LIN {X 0,Y 634.737,Z 843.139,A -85,B 0,C 180,E1 28393.414,E2 28393.414} C_VEL
LIN {X 0,Y 633.485,Z 864.639,A -85,B 0,C 180,E1 28392.949,E2 28392.949} C_VEL
LIN {X 0,Y 631.948,Z 886.443,A -85,B 0,C 180,E1 28392.362,E2 28392.362} C_VEL
LIN {X 0,Y 629.85,Z 912.243,A -85,B 0,C 180,E1 28391.511,E2 28391.511} C_VEL
LIN {X 0,Y 627.434,Z 937.199,A -85,B 0,C 180,E1 28390.495,E2 28390.495} C_VEL
LIN {X 0,Y 625.26,Z 957.685,A -85,B 0,C 180,E1 28389.527,E2 28389.527} C_VEL
LIN {X 0,Y 623.096,Z 976.739,A -85,B 0,C 180,E1 28388.507,E2 28388.507} C_VEL
LIN {X 0,Y 620.859,Z 995.438,A -85,B 0,C 180,E1 28387.383,E2 28387.383} C_VEL
LIN {X 0,Y 618.34,Z 1015.935,A -85,B 0,C 180,E1 28386,E2 28386} C_VEL
LIN {X 0,Y 615.314,Z 1039.357,A -85,B 0,C 180,E1 28384.195,E2 28384.195} C_VEL
LIN {X 0,Y 612.99,Z 1057.389,A -85,B 0,C 180,E1 28382.621,E2 28382.621} C_VEL
LIN {X 0,Y 610.906,Z 1073.81,A -85,B 0,C 180,E1 28381.035,E2 28381.035} C_VEL
LIN {X 0,Y 608.727,Z 1091.946,A -85,B 0,C 180,E1 28379.089,E2 28379.089} C_VEL
LIN {X 0,Y 606.52,Z 1110.307,A -85,B 0,C 180,E1 28376.852,E2 28376.852} C_VEL
LIN {X 0,Y 604.947,Z 1124.916,A -85,B 0,C 180,E1 28374.848,E2 28374.848} C_VEL
LIN {X 0,Y 603.439,Z 1140.182,A -85,B 0,C 180,E1 28372.504,E2 28372.504} C_VEL
LIN {X 0,Y 602.196,Z 1154.243,A -85,B 0,C 180,E1 28370.001,E2 28370.001} C_VEL
LIN {X 0,Y 601.435,Z 1164.532,A -85,B 0,C 180,E1 28367.912,E2 28367.912} C_VEL
LIN {X 0,Y 600.808,Z 1174.331,A -85,B 0,C 180,E1 28365.64,E2 28365.64} C_VEL
LIN {X 0,Y 600.353,Z 1184.273,A -85,B 0,C 180,E1 28362.895,E2 28362.895} C_VEL
LIN {X 0,Y 600.109,Z 1191.1,A -85,B 0,C 180,E1 28360.561,E2 28360.561} C_VEL
LIN {X 0,Y 599.988,Z 1196.552,A -85,B 0,C 180,E1 28358.24,E2 28358.24} C_VEL
LIN {X 0,Y 599.931,Z 1201.053,A -85,B 0,C 180,E1 28355.643,E2 28355.643} C_VEL
LIN {X 0,Y 599.918,Z 1203.723,A -85,B 0,C 180,E1 28353.153,E2 28353.153} C_VEL
LIN {X 0,Y 599.912,Z 1204.759,A -85,B 0,C 180,E1 28351.051,E2 28351.051} C_VEL
LIN {X 0,Y 599.908,Z 1204.782,A -85,B 0,C 180,E1 28349.045,E2 28349.045} C_VEL
LIN {X 0,Y 599.918,Z 1203.791,A -85,B 0,C 180,E1 28346.943,E2 28346.943} C_VEL
LIN {X 0,Y 599.93,Z 1201.177,A -85,B 0,C 180,E1 28344.453,E2 28344.453} C_VEL
LIN {X 0,Y 599.985,Z 1196.758,A -85,B 0,C 180,E1 28341.857,E2 28341.857} C_VEL
LIN {X 0,Y 600.104,Z 1191.355,A -85,B 0,C 180,E1 28339.537,E2 28339.537} C_VEL
LIN {X 0,Y 600.338,Z 1184.575,A -85,B 0,C 180,E1 28337.202,E2 28337.202} C_VEL
LIN {X 0,Y 600.787,Z 1174.735,A -85,B 0,C 180,E1 28334.458,E2 28334.458} C_VEL
LIN {X 0,Y 601.405,Z 1164.995,A -85,B 0,C 180,E1 28332.187,E2 28332.187} C_VEL
LIN {X 0,Y 602.16,Z 1154.762,A -85,B 0,C 180,E1 28330.099,E2 28330.099} C_VEL
LIN {X 0,Y 603.269,Z 1141.958,A -85,B 0,C 180,E1 28327.797,E2 28327.797} C_VEL
LIN {X 0,Y 604.785,Z 1126.491,A -85,B 0,C 180,E1 28325.379,E2 28325.379} C_VEL
LIN {X 0,Y 606.34,Z 1111.848,A -85,B 0,C 180,E1 28323.351,E2 28323.351} C_VEL
LIN {X 0,Y 608.291,Z 1095.443,A -85,B 0,C 180,E1 28321.317,E2 28321.317} C_VEL
LIN {X 0,Y 610.668,Z 1075.839,A -85,B 0,C 180,E1 28319.171,E2 28319.171} C_VEL
LIN {X 0,Y 612.801,Z 1058.916,A -85,B 0,C 180,E1 28317.52,E2 28317.52} C_VEL
LIN {X 0,Y 615.004,Z 1041.616,A -85,B 0,C 180,E1 28315.995,E2 28315.995} C_VEL
LIN {X 0,Y 617.903,Z 1019.546,A -85,B 0,C 180,E1 28314.257,E2 28314.257} C_VEL
LIN {X 0,Y 620.763,Z 996.244,A -85,B 0,C 180,E1 28312.669,E2 28312.669} C_VEL
LIN {X 0,Y 622.991,Z 977.642,A -85,B 0,C 180,E1 28311.544,E2 28311.544} C_VEL
LIN {X 0,Y 625.147,Z 958.697,A -85,B 0,C 180,E1 28310.524,E2 28310.524} C_VEL
LIN {X 0,Y 627.185,Z 939.467,A -85,B 0,C 180,E1 28309.606,E2 28309.606} C_VEL
LIN {X 0,Y 629.333,Z 917.449,A -85,B 0,C 180,E1 28308.69,E2 28308.69} C_VEL
LIN {X 0,Y 631.745,Z 889.26,A -85,B 0,C 180,E1 28307.721,E2 28307.721} C_VEL
LIN {X 0,Y 633.4,Z 865.996,A -85,B 0,C 180,E1 28307.084,E2 28307.084} C_VEL
LIN {X 0,Y 634.659,Z 844.673,A -85,B 0,C 180,E1 28306.616,E2 28306.616} C_VEL
LIN {X 0,Y 635.658,Z 822.464,A -85,B 0,C 180,E1 28306.243,E2 28306.243} C_VEL
LIN {X 0,Y 639.154,Z 652.16,A -85,B 0,C 180,E1 28303.959,E2 28303.959} C_VEL
LIN {X 0,Y 643.512,Z 444.13,A -85,B 0,C 180,E1 28301.119,E2 28301.119} C_VEL
LIN {X 0,Y 644.588,Z 389.647,A -85,B 0,C 180,E1 28300.345,E2 28300.345} C_VEL
LIN {X 0,Y 641.019,Z 373.12,A -85,B 0,C 180,E1 28299.728,E2 28299.728} C_VEL
LIN {X 0,Y 624.364,Z 349.234,A -85,B 0,C 180,E1 28297.601,E2 28297.601} C_VEL
LIN {X 0,Y 614.656,Z 330.629,A -85,B 0,C 180,E1 28295.047,E2 28295.047} C_VEL
LIN {X 0,Y 608.064,Z 317.988,A -85,B 0,C 180,E1 28293.201,E2 28293.201} C_VEL
LIN {X 0,Y 605.38,Z 313.033,A -85,B 0,C 180,E1 28292.438,E2 28292.438} C_VEL
LIN {X 0,Y 603.279,Z 308.898,A -85,B 0,C 180,E1 28291.807,E2 28291.807} C_VEL
LIN {X 0,Y 601.357,Z 305.444,A -85,B 0,C 180,E1 28291.25,E2 28291.25} C_VEL
LIN {X 0,Y 601.143,Z 304.451,A -85,B 0,C 180,E1 28291.04,E2 28291.04} C_VEL
LIN {X 0,Y 601.114,Z 304.316,A -85,B 0,C 180,E1 28287.867,E2 28287.867} C_VEL
LIN {X 0,Y 601.122,Z 304.35,A -85,B 0,C 180,E1 28284.677,E2 28284.677} C_VEL
LIN {X 0,Y 601.115,Z 304.302,A -85,B 0,C 180,E1 28281.466,E2 28281.466} C_VEL
LIN {X 0,Y 601.127,Z 304.348,A -85,B 0,C 180,E1 28278.241,E2 28278.241} C_VEL
LIN {X 0,Y 601.129,Z 304.305,A -85,B 0,C 180,E1 28274.9,E2 28274.9} C_VEL
LIN {X 0,Y 601.127,Z 304.334,A -85,B 0,C 180,E1 28271.611,E2 28271.611} C_VEL
LIN {X 0,Y 601.11,Z 304.31,A -85,B 0,C 180,E1 28268.417,E2 28268.417} C_VEL
LIN {X 0,Y 601.125,Z 304.346,A -85,B 0,C 180,E1 28265.249,E2 28265.249} C_VEL
LIN {X 0,Y 601.113,Z 304.347,A -85,B 0,C 180,E1 28262.097,E2 28262.097} C_VEL
LIN {X 0,Y 601.129,Z 304.354,A -85,B 0,C 180,E1 28258.952,E2 28258.952} C_VEL
LIN {X 0,Y 601.111,Z 304.352,A -85,B 0,C 180,E1 28255.803,E2 28255.803} C_VEL
LIN {X 0,Y 601.138,Z 304.349,A -85,B 0,C 180,E1 28252.545,E2 28252.545} C_VEL
LIN {X 0,Y 601.128,Z 304.345,A -85,B 0,C 180,E1 28249.263,E2 28249.263} C_VEL
LIN {X 0,Y 601.112,Z 304.346,A -85,B 0,C 180,E1 28246.043,E2 28246.043} C_VEL
LIN {X 0,Y 601.134,Z 304.335,A -85,B 0,C 180,E1 28242.878,E2 28242.878} C_VEL
LIN {X 0,Y 601.099,Z 304.343,A -85,B 0,C 180,E1 28239.656,E2 28239.656} C_VEL
LIN {X 0,Y 601.134,Z 304.327,A -85,B 0,C 180,E1 28236.575,E2 28236.575} C_VEL
LIN {X 0,Y 601.094,Z 304.318,A -85,B 0,C 180,E1 28233.418,E2 28233.418} C_VEL
LIN {X 0,Y 601.135,Z 304.326,A -85,B 0,C 180,E1 28230.254,E2 28230.254} C_VEL
LIN {X 0,Y 601.092,Z 304.325,A -85,B 0,C 180,E1 28227.142,E2 28227.142} C_VEL
LIN {X 0,Y 601.126,Z 304.31,A -85,B 0,C 180,E1 28223.926,E2 28223.926} C_VEL
LIN {X 0,Y 601.099,Z 304.355,A -85,B 0,C 180,E1 28220.794,E2 28220.794} C_VEL
LIN {X 0,Y 601.098,Z 304.309,A -85,B 0,C 180,E1 28217.466,E2 28217.466} C_VEL
LIN {X 0,Y 601.112,Z 304.544,A -85,B 0,C 180,E1 28214.878,E2 28214.878} C_VEL
LIN {X 0,Y 602.437,Z 307.817,A -85,B 0,C 180,E1 28214.325,E2 28214.325} C_VEL
LIN {X 0,Y 603.781,Z 310.243,A -85,B 0,C 180,E1 28213.914,E2 28213.914} C_VEL
LIN {X 0,Y 610.058,Z 322.832,A -85,B 0,C 180,E1 28211.917,E2 28211.917} C_VEL
LIN {X 0,Y 618.337,Z 340.119,A -85,B 0,C 180,E1 28209.379,E2 28209.379} C_VEL
LIN {X 0,Y 621.916,Z 347.601,A -85,B 0,C 180,E1 28208.371,E2 28208.371} C_VEL
LIN {X 0,Y 634.739,Z 366.423,A -85,B 0,C 180,E1 28206.763,E2 28206.763} C_VEL
LIN {X 0,Y 635.552,Z 368.337,A -85,B 0,C 180,E1 28206.653,E2 28206.653} C_VEL
LIN {X 0,Y 635.77,Z 369.283,A -85,B 0,C 180,E1 28206.616,E2 28206.616} C_VEL
LIN {X 0,Y 636.509,Z 375.596,A -85,B 0,C 180,E1 28206.442,E2 28206.442} C_VEL
LIN {X 0,Y 635.968,Z 384.479,A -85,B 0,C 180,E1 28206.352,E2 28206.352} C_VEL
LIN {X 0,Y 633.615,Z 401.55,A -85,B 0,C 180,E1 28206.306,E2 28206.306} C_VEL
LIN {X 0,Y 633.425,Z 404.97,A -85,B 0,C 180,E1 28206.27,E2 28206.27} C_VEL
LIN {X 0,Y 627.887,Z 630.342,A -85,B 0,C 180,E1 28203.198,E2 28203.198} C_VEL
LIN {X 0,Y 624.144,Z 782.263,A -85,B 0,C 180,E1 28201.133,E2 28201.133} C_VEL
LIN {X 0,Y 622.848,Z 808.88,A -85,B 0,C 180,E1 28200.626,E2 28200.626} C_VEL
LIN {X 0,Y 621.288,Z 831.683,A -85,B 0,C 180,E1 28200.033,E2 28200.033} C_VEL
LIN {X 0,Y 619.625,Z 852.177,A -85,B 0,C 180,E1 28199.377,E2 28199.377} C_VEL
LIN {X 0,Y 617.403,Z 876.604,A -85,B 0,C 180,E1 28198.43,E2 28198.43} C_VEL
LIN {X 0,Y 615.001,Z 898.626,A -85,B 0,C 180,E1 28197.393,E2 28197.393} C_VEL
LIN {X 0,Y 612.877,Z 916.885,A -85,B 0,C 180,E1 28196.404,E2 28196.404} C_VEL
LIN {X 0,Y 610.566,Z 935.623,A -85,B 0,C 180,E1 28195.251,E2 28195.251} C_VEL
LIN {X 0,Y 607.657,Z 957.975,A -85,B 0,C 180,E1 28193.671,E2 28193.671} C_VEL
LIN {X 0,Y 604.491,Z 983.088,A -85,B 0,C 180,E1 28191.626,E2 28191.626} C_VEL
LIN {X 0,Y 602.054,Z 1002.514,A -85,B 0,C 180,E1 28189.803,E2 28189.803} C_VEL
LIN {X 0,Y 600.17,Z 1018.198,A -85,B 0,C 180,E1 28188.152,E2 28188.152} C_VEL
LIN {X 0,Y 598.217,Z 1035.5,A -85,B 0,C 180,E1 28186.108,E2 28186.108} C_VEL
LIN {X 0,Y 596.541,Z 1050.571,A -85,B 0,C 180,E1 28184.066,E2 28184.066} C_VEL
LIN {X 0,Y 595.307,Z 1063.353,A -85,B 0,C 180,E1 28182.119,E2 28182.119} C_VEL
LIN {X 0,Y 594.083,Z 1077.311,A -85,B 0,C 180,E1 28179.689,E2 28179.689} C_VEL
LIN {X 0,Y 593.289,Z 1087.834,A -85,B 0,C 180,E1 28177.553,E2 28177.553} C_VEL
LIN {X 0,Y 592.738,Z 1096.969,A -85,B 0,C 180,E1 28175.42,E2 28175.42} C_VEL
LIN {X 0,Y 592.306,Z 1106.272,A -85,B 0,C 180,E1 28172.806,E2 28172.806} C_VEL
LIN {X 0,Y 592.077,Z 1112.145,A -85,B 0,C 180,E1 28170.774,E2 28170.774} C_VEL
LIN {X 0,Y 591.987,Z 1116.904,A -85,B 0,C 180,E1 28168.742,E2 28168.742} C_VEL
LIN {X 0,Y 591.917,Z 1121.208,A -85,B 0,C 180,E1 28166.32,E2 28166.32} C_VEL
LIN {X 0,Y 591.912,Z 1123.779,A -85,B 0,C 180,E1 28163.891,E2 28163.891} C_VEL
LIN {X 0,Y 591.915,Z 1124.8,A -85,B 0,C 180,E1 28161.843,E2 28161.843} C_VEL
LIN {X 0,Y 591.904,Z 1124.734,A -85,B 0,C 180,E1 28159.783,E2 28159.783} C_VEL
LIN {X 0,Y 591.918,Z 1123.242,A -85,B 0,C 180,E1 28157.315,E2 28157.315} C_VEL
LIN {X 0,Y 591.921,Z 1120.275,A -85,B 0,C 180,E1 28155.022,E2 28155.022} C_VEL
LIN {X 0,Y 591.988,Z 1116.421,A -85,B 0,C 180,E1 28152.941,E2 28152.941} C_VEL
LIN {X 0,Y 592.112,Z 1111.473,A -85,B 0,C 180,E1 28150.877,E2 28150.877} C_VEL
LIN {X 0,Y 592.395,Z 1103.669,A -85,B 0,C 180,E1 28148.307,E2 28148.307} C_VEL
LIN {X 0,Y 592.828,Z 1095.329,A -85,B 0,C 180,E1 28146.088,E2 28146.088} C_VEL
LIN {X 0,Y 593.414,Z 1086.275,A -85,B 0,C 180,E1 28144.018,E2 28144.018} C_VEL
LIN {X 0,Y 594.431,Z 1073.185,A -85,B 0,C 180,E1 28141.465,E2 28141.465} C_VEL
LIN {X 0,Y 595.521,Z 1061.026,A -85,B 0,C 180,E1 28139.421,E2 28139.421} C_VEL
LIN {X 0,Y 596.932,Z 1047.21,A -85,B 0,C 180,E1 28137.361,E2 28137.361} C_VEL
LIN {X 0,Y 598.756,Z 1030.354,A -85,B 0,C 180,E1 28135.173,E2 28135.173} C_VEL
LIN {X 0,Y 600.547,Z 1015.057,A -85,B 0,C 180,E1 28133.413,E2 28133.413} C_VEL
LIN {X 0,Y 602.877,Z 996.133,A -85,B 0,C 180,E1 28131.476,E2 28131.476} C_VEL
LIN {X 0,Y 605.186,Z 976.858,A -85,B 0,C 180,E1 28129.758,E2 28129.758} C_VEL
LIN {X 0,Y 608.508,Z 951.843,A -85,B 0,C 180,E1 28127.775,E2 28127.775} C_VEL
LIN {X 0,Y 610.992,Z 932.614,A -85,B 0,C 180,E1 28126.453,E2 28126.453} C_VEL
LIN {X 0,Y 613.37,Z 913.498,A -85,B 0,C 180,E1 28125.296,E2 28125.296} C_VEL
LIN {X 0,Y 616.143,Z 889.259,A -85,B 0,C 180,E1 28124.037,E2 28124.037} C_VEL
LIN {X 0,Y 618.322,Z 867.895,A -85,B 0,C 180,E1 28123.105,E2 28123.105} C_VEL
LIN {X 0,Y 620.368,Z 845.635,A -85,B 0,C 180,E1 28122.287,E2 28122.287} C_VEL
LIN {X 0,Y 622.332,Z 819.853,A -85,B 0,C 180,E1 28121.532,E2 28121.532} C_VEL
LIN {X 0,Y 623.576,Z 798.797,A -85,B 0,C 180,E1 28121.052,E2 28121.052} C_VEL
LIN {X 0,Y 624.552,Z 776.726,A -85,B 0,C 180,E1 28120.672,E2 28120.672} C_VEL
LIN {X 0,Y 630.566,Z 536.64,A -85,B 0,C 180,E1 28117.405,E2 28117.405} C_VEL
LIN {X 0,Y 634.45,Z 387.315,A -85,B 0,C 180,E1 28115.324,E2 28115.324} C_VEL
LIN {X 0,Y 631.23,Z 372.127,A -85,B 0,C 180,E1 28114.713,E2 28114.713} C_VEL
LIN {X 0,Y 621.138,Z 357.085,A -85,B 0,C 180,E1 28113.294,E2 28113.294} C_VEL
LIN {X 0,Y 614.055,Z 346.626,A -85,B 0,C 180,E1 28112.172,E2 28112.172} C_VEL
LIN {X 0,Y 607.583,Z 333.131,A -85,B 0,C 180,E1 28109.91,E2 28109.91} C_VEL
LIN {X 0,Y 602.57,Z 323.528,A -85,B 0,C 180,E1 28108.116,E2 28108.116} C_VEL
LIN {X 0,Y 600.308,Z 319.191,A -85,B 0,C 180,E1 28107.261,E2 28107.261} C_VEL
LIN {X 0,Y 597.846,Z 314.566,A -85,B 0,C 180,E1 28106.308,E2 28106.308} C_VEL
LIN {X 0,Y 595.889,Z 310.557,A -85,B 0,C 180,E1 28105.482,E2 28105.482} C_VEL
LIN {X 0,Y 593.523,Z 306.861,A -85,B 0,C 180,E1 28104.59,E2 28104.59} C_VEL
LIN {X 0,Y 593.205,Z 305.46,A -85,B 0,C 180,E1 28104.235,E2 28104.235} C_VEL
LIN {X 0,Y 593.187,Z 305.301,A -85,B 0,C 180,E1 28100.938,E2 28100.938} C_VEL
LIN {X 0,Y 593.186,Z 305.3,A -85,B 0,C 180,E1 28097.759,E2 28097.759} C_VEL
LIN {X 0,Y 593.181,Z 305.343,A -85,B 0,C 180,E1 28094.546,E2 28094.546} C_VEL
LIN {X 0,Y 593.18,Z 305.301,A -85,B 0,C 180,E1 28091.375,E2 28091.375} C_VEL
LIN {X 0,Y 593.176,Z 305.313,A -85,B 0,C 180,E1 28088.238,E2 28088.238} C_VEL
LIN {X 0,Y 593.18,Z 305.328,A -85,B 0,C 180,E1 28085.029,E2 28085.029} C_VEL
LIN {X 0,Y 593.179,Z 305.295,A -85,B 0,C 180,E1 28081.835,E2 28081.835} C_VEL
LIN {X 0,Y 593.193,Z 305.339,A -85,B 0,C 180,E1 28078.551,E2 28078.551} C_VEL
LIN {X 0,Y 593.184,Z 305.298,A -85,B 0,C 180,E1 28075.262,E2 28075.262} C_VEL
LIN {X 0,Y 593.186,Z 305.314,A -85,B 0,C 180,E1 28072.055,E2 28072.055} C_VEL
LIN {X 0,Y 593.178,Z 305.326,A -85,B 0,C 180,E1 28068.818,E2 28068.818} C_VEL
LIN {X 0,Y 593.18,Z 305.296,A -85,B 0,C 180,E1 28065.653,E2 28065.653} C_VEL
LIN {X 0,Y 593.178,Z 305.34,A -85,B 0,C 180,E1 28062.438,E2 28062.438} C_VEL
LIN {X 0,Y 593.19,Z 305.307,A -85,B 0,C 180,E1 28059.166,E2 28059.166} C_VEL
LIN {X 0,Y 593.186,Z 305.296,A -85,B 0,C 180,E1 28055.926,E2 28055.926} C_VEL
LIN {X 0,Y 593.181,Z 305.318,A -85,B 0,C 180,E1 28052.601,E2 28052.601} C_VEL
LIN {X 0,Y 593.233,Z 305.627,A -85,B 0,C 180,E1 28051.214,E2 28051.214} C_VEL
LIN {X 0,Y 594.731,Z 309.137,A -85,B 0,C 180,E1 28050.488,E2 28050.488} C_VEL
LIN {X 0,Y 596.204,Z 311.055,A -85,B 0,C 180,E1 28050.015,E2 28050.015} C_VEL
LIN {X 0,Y 598.26,Z 314.959,A -85,B 0,C 180,E1 28049.241,E2 28049.241} C_VEL
LIN {X 0,Y 599.372,Z 316.945,A -85,B 0,C 180,E1 28048.845,E2 28048.845} C_VEL
LIN {X 0,Y 602.237,Z 322.081,A -85,B 0,C 180,E1 28047.857,E2 28047.857} C_VEL
LIN {X 0,Y 605.079,Z 327.328,A -85,B 0,C 180,E1 28046.907,E2 28046.907} C_VEL
LIN {X 0,Y 609.467,Z 335.318,A -85,B 0,C 180,E1 28045.528,E2 28045.528} C_VEL
LIN {X 0,Y 615.852,Z 348.153,A -85,B 0,C 180,E1 28043.542,E2 28043.542} C_VEL
LIN {X 0,Y 617.493,Z 350.954,A -85,B 0,C 180,E1 28043.192,E2 28043.192} C_VEL
LIN {X 0,Y 633.776,Z 374.667,A -85,B 0,C 180,E1 28040.944,E2 28040.944} C_VEL
LIN {X 0,Y 636.298,Z 378.781,A -85,B 0,C 180,E1 28040.613,E2 28040.613} C_VEL
LIN {X 0,Y 639.01,Z 393.151,A -85,B 0,C 180,E1 28040.1,E2 28040.1} C_VEL
LIN {X 0,Y 634.195,Z 606.611,A -85,B 0,C 180,E1 28037.148,E2 28037.148} C_VEL
LIN {X 0,Y 629.632,Z 823.84,A -85,B 0,C 180,E1 28034.222,E2 28034.222} C_VEL
LIN {X 0,Y 628.645,Z 846.019,A -85,B 0,C 180,E1 28033.849,E2 28033.849} C_VEL
LIN {X 0,Y 627.348,Z 868.333,A -85,B 0,C 180,E1 28033.359,E2 28033.359} C_VEL
LIN {X 0,Y 625.389,Z 894.349,A -85,B 0,C 180,E1 28032.622,E2 28032.622} C_VEL
LIN {X 0,Y 623.049,Z 919.238,A -85,B 0,C 180,E1 28031.733,E2 28031.733} C_VEL
LIN {X 0,Y 620.978,Z 939.457,A -85,B 0,C 180,E1 28030.883,E2 28030.883} C_VEL
LIN {X 0,Y 618.822,Z 958.686,A -85,B 0,C 180,E1 28029.96,E2 28029.96} C_VEL
LIN {X 0,Y 616.544,Z 977.636,A -85,B 0,C 180,E1 28028.933,E2 28028.933} C_VEL
LIN {X 0,Y 614.088,Z 997.058,A -85,B 0,C 180,E1 28027.749,E2 28027.749} C_VEL
LIN {X 0,Y 610.965,Z 1020.889,A -85,B 0,C 180,E1 28026.097,E2 28026.097} C_VEL
LIN {X 0,Y 608.094,Z 1041.617,A -85,B 0,C 180,E1 28024.446,E2 28024.446} C_VEL
LIN {X 0,Y 605.719,Z 1059.052,A -85,B 0,C 180,E1 28022.894,E2 28022.894} C_VEL
LIN {X 0,Y 603.289,Z 1077.265,A -85,B 0,C 180,E1 28021.092,E2 28021.092} C_VEL
LIN {X 0,Y 600.702,Z 1097.146,A -85,B 0,C 180,E1 28018.862,E2 28018.862} C_VEL
LIN {X 0,Y 598.746,Z 1112.644,A -85,B 0,C 180,E1 28016.903,E2 28016.903} C_VEL
LIN {X 0,Y 597.075,Z 1127.449,A -85,B 0,C 180,E1 28014.815,E2 28014.815} C_VEL
LIN {X 0,Y 595.364,Z 1143.703,A -85,B 0,C 180,E1 28012.202,E2 28012.202} C_VEL
LIN {X 0,Y 594.298,Z 1155.27,A -85,B 0,C 180,E1 28010.073,E2 28010.073} C_VEL
LIN {X 0,Y 593.5,Z 1165.448,A -85,B 0,C 180,E1 28007.957,E2 28007.957} C_VEL
LIN {X 0,Y 592.788,Z 1176.306,A -85,B 0,C 180,E1 28005.356,E2 28005.356} C_VEL
LIN {X 0,Y 592.348,Z 1185.179,A -85,B 0,C 180,E1 28002.775,E2 28002.775} C_VEL
LIN {X 0,Y 592.108,Z 1191.86,A -85,B 0,C 180,E1 28000.41,E2 28000.41} C_VEL
LIN {X 0,Y 591.981,Z 1197.542,A -85,B 0,C 180,E1 27997.863,E2 27997.863} C_VEL
LIN {X 0,Y 591.928,Z 1201.66,A -85,B 0,C 180,E1 27995.234,E2 27995.234} C_VEL
LIN {X 0,Y 591.915,Z 1203.925,A -85,B 0,C 180,E1 27992.905,E2 27992.905} C_VEL
LIN {X 0,Y 591.895,Z 1204.849,A -85,B 0,C 180,E1 27990.678,E2 27990.678} C_VEL
LIN {X 0,Y 591.908,Z 1204.623,A -85,B 0,C 180,E1 27988.355,E2 27988.355} C_VEL
LIN {X 0,Y 591.918,Z 1202.789,A -85,B 0,C 180,E1 27985.738,E2 27985.738} C_VEL
LIN {X 0,Y 591.944,Z 1199.546,A -85,B 0,C 180,E1 27983.307,E2 27983.307} C_VEL
LIN {X 0,Y 592.022,Z 1195.103,A -85,B 0,C 180,E1 27980.963,E2 27980.963} C_VEL
LIN {X 0,Y 592.224,Z 1188.471,A -85,B 0,C 180,E1 27978.31,E2 27978.31} C_VEL
LIN {X 0,Y 592.556,Z 1180.571,A -85,B 0,C 180,E1 27975.838,E2 27975.838} C_VEL
LIN {X 0,Y 593.028,Z 1172.305,A -85,B 0,C 180,E1 27973.646,E2 27973.646} C_VEL
LIN {X 0,Y 593.709,Z 1162.694,A -85,B 0,C 180,E1 27971.44,E2 27971.44} C_VEL
LIN {X 0,Y 594.841,Z 1149.447,A -85,B 0,C 180,E1 27968.815,E2 27968.815} C_VEL
LIN {X 0,Y 596.107,Z 1136.315,A -85,B 0,C 180,E1 27966.567,E2 27966.567} C_VEL
LIN {X 0,Y 597.54,Z 1122.985,A -85,B 0,C 180,E1 27964.53,E2 27964.53} C_VEL
LIN {X 0,Y 599.573,Z 1106.413,A -85,B 0,C 180,E1 27962.273,E2 27962.273} C_VEL
LIN {X 0,Y 601.819,Z 1088.229,A -85,B 0,C 180,E1 27960.105,E2 27960.105} C_VEL
LIN {X 0,Y 603.941,Z 1072.291,A -85,B 0,C 180,E1 27958.4,E2 27958.4} C_VEL
LIN {X 0,Y 606.351,Z 1054.613,A -85,B 0,C 180,E1 27956.694,E2 27956.694} C_VEL
LIN {X 0,Y 609.496,Z 1031.566,A -85,B 0,C 180,E1 27954.729,E2 27954.729} C_VEL
LIN {X 0,Y 612.158,Z 1011.517,A -85,B 0,C 180,E1 27953.229,E2 27953.229} C_VEL
LIN {X 0,Y 614.692,Z 992.1,A -85,B 0,C 180,E1 27951.934,E2 27951.934} C_VEL
LIN {X 0,Y 617.675,Z 968.571,A -85,B 0,C 180,E1 27950.549,E2 27950.549} C_VEL
LIN {X 0,Y 620.471,Z 943.985,A -85,B 0,C 180,E1 27949.32,E2 27949.32} C_VEL
LIN {X 0,Y 622.709,Z 922.583,A -85,B 0,C 180,E1 27948.399,E2 27948.399} C_VEL
LIN {X 0,Y 624.663,Z 901.901,A -85,B 0,C 180,E1 27947.634,E2 27947.634} C_VEL
LIN {X 0,Y 626.529,Z 879.6,A -85,B 0,C 180,E1 27946.939,E2 27946.939} C_VEL
LIN {X 0,Y 628.34,Z 852.631,A -85,B 0,C 180,E1 27946.278,E2 27946.278} C_VEL
LIN {X 0,Y 629.539,Z 827.007,A -85,B 0,C 180,E1 27945.822,E2 27945.822} C_VEL
LIN {X 0,Y 632.652,Z 684.755,A -85,B 0,C 180,E1 27943.901,E2 27943.901} C_VEL
LIN {X 0,Y 637.392,Z 469.924,A -85,B 0,C 180,E1 27940.958,E2 27940.958} C_VEL
LIN {X 0,Y 639.12,Z 391.738,A -85,B 0,C 180,E1 27939.848,E2 27939.848} C_VEL
LIN {X 0,Y 636.184,Z 378.113,A -85,B 0,C 180,E1 27939.33,E2 27939.33} C_VEL
LIN {X 0,Y 616.066,Z 349.467,A -85,B 0,C 180,E1 27936.733,E2 27936.733} C_VEL
LIN {X 0,Y 606.711,Z 331.431,A -85,B 0,C 180,E1 27934.193,E2 27934.193} C_VEL
LIN {X 0,Y 599.863,Z 318.515,A -85,B 0,C 180,E1 27932.235,E2 27932.235} C_VEL
LIN {X 0,Y 597.671,Z 314.326,A -85,B 0,C 180,E1 27931.577,E2 27931.577} C_VEL
LIN {X 0,Y 595.189,Z 309.685,A -85,B 0,C 180,E1 27930.823,E2 27930.823} C_VEL
LIN {X 0,Y 593.374,Z 306.265,A -85,B 0,C 180,E1 27930.255,E2 27930.255} C_VEL
LIN {X 0,Y 593.197,Z 305.427,A -85,B 0,C 180,E1 27930.041,E2 27930.041} C_VEL
LIN {X 0,Y 593.181,Z 305.29,A -85,B 0,C 180,E1 27926.856,E2 27926.856} C_VEL
LIN {X 0,Y 593.179,Z 305.331,A -85,B 0,C 180,E1 27923.652,E2 27923.652} C_VEL
LIN {X 0,Y 593.178,Z 305.302,A -85,B 0,C 180,E1 27920.525,E2 27920.525} C_VEL
LIN {X 0,Y 593.18,Z 305.306,A -85,B 0,C 180,E1 27917.359,E2 27917.359} C_VEL
LIN {X 0,Y 593.181,Z 305.315,A -85,B 0,C 180,E1 27914.148,E2 27914.148} C_VEL
LIN {X 0,Y 593.187,Z 305.297,A -85,B 0,C 180,E1 27910.882,E2 27910.882} C_VEL
LIN {X 0,Y 593.192,Z 305.324,A -85,B 0,C 180,E1 27907.555,E2 27907.555} C_VEL
LIN {X 0,Y 593.176,Z 305.33,A -85,B 0,C 180,E1 27904.35,E2 27904.35} C_VEL
LIN {X 0,Y 593.187,Z 305.328,A -85,B 0,C 180,E1 27901.159,E2 27901.159} C_VEL
LIN {X 0,Y 593.17,Z 305.328,A -85,B 0,C 180,E1 27897.971,E2 27897.971} C_VEL
LIN {X 0,Y 593.194,Z 305.332,A -85,B 0,C 180,E1 27894.681,E2 27894.681} C_VEL
LIN {X 0,Y 593.181,Z 305.337,A -85,B 0,C 180,E1 27891.469,E2 27891.469} C_VEL
LIN {X 0,Y 593.177,Z 305.34,A -85,B 0,C 180,E1 27888.132,E2 27888.132} C_VEL
LIN {X 0,Y 593.2,Z 305.338,A -85,B 0,C 180,E1 27884.955,E2 27884.955} C_VEL
LIN {X 0,Y 593.164,Z 305.344,A -85,B 0,C 180,E1 27881.727,E2 27881.727} C_VEL
LIN {X 0,Y 593.199,Z 305.336,A -85,B 0,C 180,E1 27878.499,E2 27878.499} C_VEL
LIN {X 0,Y 593.152,Z 305.29,A -85,B 0,C 180,E1 27875.394,E2 27875.394} C_VEL
LIN {X 0,Y 593.2,Z 305.333,A -85,B 0,C 180,E1 27872.166,E2 27872.166} C_VEL
LIN {X 0,Y 593.157,Z 305.291,A -85,B 0,C 180,E1 27869.06,E2 27869.06} C_VEL
LIN {X 0,Y 593.175,Z 305.345,A -85,B 0,C 180,E1 27865.736,E2 27865.736} C_VEL
LIN {X 0,Y 593.179,Z 305.289,A -85,B 0,C 180,E1 27862.553,E2 27862.553} C_VEL
LIN {X 0,Y 593.153,Z 305.317,A -85,B 0,C 180,E1 27859.336,E2 27859.336} C_VEL
LIN {X 0,Y 593.197,Z 305.323,A -85,B 0,C 180,E1 27856.149,E2 27856.149} C_VEL
LIN {X 0,Y 593.268,Z 305.827,A -85,B 0,C 180,E1 27855.753,E2 27855.753} C_VEL
LIN {X 0,Y 594.698,Z 309.158,A -85,B 0,C 180,E1 27855.194,E2 27855.194} C_VEL
LIN {X 0,Y 595.935,Z 311.517,A -85,B 0,C 180,E1 27854.787,E2 27854.787} C_VEL
LIN {X 0,Y 598.222,Z 315.85,A -85,B 0,C 180,E1 27854.051,E2 27854.051} C_VEL
LIN {X 0,Y 604.443,Z 328.451,A -85,B 0,C 180,E1 27852.033,E2 27852.033} C_VEL
LIN {X 0,Y 612.463,Z 345.252,A -85,B 0,C 180,E1 27849.545,E2 27849.545} C_VEL
LIN {X 0,Y 613.838,Z 347.799,A -85,B 0,C 180,E1 27849.217,E2 27849.217} C_VEL
LIN {X 0,Y 629.897,Z 371.21,A -85,B 0,C 180,E1 27847.167,E2 27847.167} C_VEL
LIN {X 0,Y 630.758,Z 373.41,A -85,B 0,C 180,E1 27847.045,E2 27847.045} C_VEL
LIN {X 0,Y 633.841,Z 388.559,A -85,B 0,C 180,E1 27846.494,E2 27846.494} C_VEL
LIN {X 0,Y 633.425,Z 404.97,A -85,B 0,C 180,E1 27846.27,E2 27846.27} C_VEL
LIN {X 0,Y 632.552,Z 412.675,A -85,B 0,C 180,E1 27846.23,E2 27846.23} C_VEL
LIN {X 0,Y 627.751,Z 433.322,A -85,B 0,C 180,E1 27846.364,E2 27846.364} C_VEL
LIN {X 0,Y 627.068,Z 439.932,A -85,B 0,C 180,E1 27846.324,E2 27846.324} C_VEL
LIN {X 0,Y 621.351,Z 664.116,A -85,B 0,C 180,E1 27843.259,E2 27843.259} C_VEL
LIN {X 0,Y 618.257,Z 782.871,A -85,B 0,C 180,E1 27841.63,E2 27841.63} C_VEL
LIN {X 0,Y 616.874,Z 809.805,A -85,B 0,C 180,E1 27841.111,E2 27841.111} C_VEL
LIN {X 0,Y 615.261,Z 832.313,A -85,B 0,C 180,E1 27840.52,E2 27840.52} C_VEL
LIN {X 0,Y 613.517,Z 852.781,A -85,B 0,C 180,E1 27839.86,E2 27839.86} C_VEL
LIN {X 0,Y 611.188,Z 877.138,A -85,B 0,C 180,E1 27838.909,E2 27838.909} C_VEL
LIN {X 0,Y 608.663,Z 899.206,A -85,B 0,C 180,E1 27837.862,E2 27837.862} C_VEL
LIN {X 0,Y 606.412,Z 917.602,A -85,B 0,C 180,E1 27836.857,E2 27836.857} C_VEL
LIN {X 0,Y 603.904,Z 936.945,A -85,B 0,C 180,E1 27835.655,E2 27835.655} C_VEL
LIN {X 0,Y 600.726,Z 959.903,A -85,B 0,C 180,E1 27834.003,E2 27834.003} C_VEL
LIN {X 0,Y 598.217,Z 977.418,A -85,B 0,C 180,E1 27832.556,E2 27832.556} C_VEL
LIN {X 0,Y 595.281,Z 998.952,A -85,B 0,C 180,E1 27830.551,E2 27830.551} C_VEL
LIN {X 0,Y 593.082,Z 1015.822,A -85,B 0,C 180,E1 27828.784,E2 27828.784} C_VEL
LIN {X 0,Y 591.192,Z 1030.97,A -85,B 0,C 180,E1 27827.013,E2 27827.013} C_VEL
LIN {X 0,Y 589.21,Z 1048.084,A -85,B 0,C 180,E1 27824.746,E2 27824.746} C_VEL
LIN {X 0,Y 587.781,Z 1061.093,A -85,B 0,C 180,E1 27822.776,E2 27822.776} C_VEL
LIN {X 0,Y 586.625,Z 1073.229,A -85,B 0,C 180,E1 27820.707,E2 27820.707} C_VEL
LIN {X 0,Y 585.533,Z 1086.182,A -85,B 0,C 180,E1 27818.148,E2 27818.148} C_VEL
LIN {X 0,Y 584.922,Z 1095.107,A -85,B 0,C 180,E1 27816.084,E2 27816.084} C_VEL
LIN {X 0,Y 584.465,Z 1103.153,A -85,B 0,C 180,E1 27813.924,E2 27813.924} C_VEL
LIN {X 0,Y 584.149,Z 1111.209,A -85,B 0,C 180,E1 27811.275,E2 27811.275} C_VEL
LIN {X 0,Y 584.002,Z 1116.344,A -85,B 0,C 180,E1 27809.117,E2 27809.117} C_VEL
LIN {X 0,Y 583.936,Z 1120.138,A -85,B 0,C 180,E1 27807.055,E2 27807.055} C_VEL
LIN {X 0,Y 583.904,Z 1123.299,A -85,B 0,C 180,E1 27804.596,E2 27804.596} C_VEL
LIN {X 0,Y 583.917,Z 1124.737,A -85,B 0,C 180,E1 27802.126,E2 27802.126} C_VEL
LIN {X 0,Y 583.897,Z 1124.797,A -85,B 0,C 180,E1 27800.04,E2 27800.04} C_VEL
LIN {X 0,Y 583.911,Z 1123.726,A -85,B 0,C 180,E1 27797.901,E2 27797.901} C_VEL
LIN {X 0,Y 583.923,Z 1120.888,A -85,B 0,C 180,E1 27795.32,E2 27795.32} C_VEL
LIN {X 0,Y 583.992,Z 1116.939,A -85,B 0,C 180,E1 27793.079,E2 27793.079} C_VEL
LIN {X 0,Y 584.109,Z 1112.194,A -85,B 0,C 180,E1 27791.02,E2 27791.02} C_VEL
LIN {X 0,Y 584.346,Z 1105.953,A -85,B 0,C 180,E1 27788.836,E2 27788.836} C_VEL
LIN {X 0,Y 584.837,Z 1096.628,A -85,B 0,C 180,E1 27786.204,E2 27786.204} C_VEL
LIN {X 0,Y 585.44,Z 1087.59,A -85,B 0,C 180,E1 27784.074,E2 27784.074} C_VEL
LIN {X 0,Y 586.331,Z 1076.704,A -85,B 0,C 180,E1 27781.844,E2 27781.844} C_VEL
LIN {X 0,Y 587.625,Z 1062.856,A -85,B 0,C 180,E1 27779.419,E2 27779.419} C_VEL
LIN {X 0,Y 588.894,Z 1050.727,A -85,B 0,C 180,E1 27777.551,E2 27777.551} C_VEL
LIN {X 0,Y 590.736,Z 1035.048,A -85,B 0,C 180,E1 27775.399,E2 27775.399} C_VEL
LIN {X 0,Y 592.834,Z 1017.755,A -85,B 0,C 180,E1 27773.341,E2 27773.341} C_VEL
LIN {X 0,Y 594.858,Z 1001.983,A -85,B 0,C 180,E1 27771.667,E2 27771.667} C_VEL
LIN {X 0,Y 598.1,Z 978.43,A -85,B 0,C 180,E1 27769.436,E2 27769.436} C_VEL
LIN {X 0,Y 600.601,Z 961.131,A -85,B 0,C 180,E1 27767.992,E2 27767.992} C_VEL
LIN {X 0,Y 603.69,Z 939.447,A -85,B 0,C 180,E1 27766.402,E2 27766.402} C_VEL
LIN {X 0,Y 606.376,Z 918.942,A -85,B 0,C 180,E1 27765.111,E2 27765.111} C_VEL
LIN {X 0,Y 608.615,Z 900.948,A -85,B 0,C 180,E1 27764.117,E2 27764.117} C_VEL
LIN {X 0,Y 610.995,Z 880.4,A -85,B 0,C 180,E1 27763.126,E2 27763.126} C_VEL
LIN {X 0,Y 613.551,Z 855.071,A -85,B 0,C 180,E1 27762.108,E2 27762.108} C_VEL
LIN {X 0,Y 615.387,Z 833.714,A -85,B 0,C 180,E1 27761.406,E2 27761.406} C_VEL
LIN {X 0,Y 616.889,Z 813.151,A -85,B 0,C 180,E1 27760.856,E2 27760.856} C_VEL
LIN {X 0,Y 618.34,Z 788.047,A -85,B 0,C 180,E1 27760.338,E2 27760.338} C_VEL
LIN {X 0,Y 619.677,Z 742.474,A -85,B 0,C 180,E1 27759.688,E2 27759.688} C_VEL
LIN {X 0,Y 626.063,Z 503.632,A -85,B 0,C 180,E1 27756.407,E2 27756.407} C_VEL
LIN {X 0,Y 629.227,Z 389.301,A -85,B 0,C 180,E1 27754.791,E2 27754.791} C_VEL
LIN {X 0,Y 626.621,Z 376.921,A -85,B 0,C 180,E1 27754.283,E2 27754.283} C_VEL
LIN {X 0,Y 614.739,Z 359.161,A -85,B 0,C 180,E1 27752.546,E2 27752.546} C_VEL
LIN {X 0,Y 606.2,Z 347.127,A -85,B 0,C 180,E1 27751.193,E2 27751.193} C_VEL
LIN {X 0,Y 600.02,Z 334.507,A -85,B 0,C 180,E1 27748.973,E2 27748.973} C_VEL
LIN {X 0,Y 594.999,Z 324.956,A -85,B 0,C 180,E1 27747.092,E2 27747.092} C_VEL
LIN {X 0,Y 592.561,Z 320.372,A -85,B 0,C 180,E1 27746.13,E2 27746.13} C_VEL
LIN {X 0,Y 590.228,Z 315.9,A -85,B 0,C 180,E1 27745.164,E2 27745.164} C_VEL
LIN {X 0,Y 588.158,Z 312.08,A -85,B 0,C 180,E1 27744.294,E2 27744.294} C_VEL
LIN {X 0,Y 585.593,Z 307.813,A -85,B 0,C 180,E1 27743.23,E2 27743.23} C_VEL
LIN {X 0,Y 585.264,Z 306.463,A -85,B 0,C 180,E1 27742.863,E2 27742.863} C_VEL
LIN {X 0,Y 585.249,Z 306.324,A -85,B 0,C 180,E1 27739.668,E2 27739.668} C_VEL
LIN {X 0,Y 585.234,Z 306.285,A -85,B 0,C 180,E1 27736.476,E2 27736.476} C_VEL
LIN {X 0,Y 585.243,Z 306.298,A -85,B 0,C 180,E1 27733.335,E2 27733.335} C_VEL
LIN {X 0,Y 585.244,Z 306.324,A -85,B 0,C 180,E1 27730.036,E2 27730.036} C_VEL
LIN {X 0,Y 585.254,Z 306.277,A -85,B 0,C 180,E1 27726.672,E2 27726.672} C_VEL
LIN {X 0,Y 585.245,Z 306.316,A -85,B 0,C 180,E1 27723.33,E2 27723.33} C_VEL
LIN {X 0,Y 585.241,Z 306.302,A -85,B 0,C 180,E1 27720.098,E2 27720.098} C_VEL
LIN {X 0,Y 585.237,Z 306.288,A -85,B 0,C 180,E1 27716.964,E2 27716.964} C_VEL
LIN {X 0,Y 585.245,Z 306.327,A -85,B 0,C 180,E1 27713.722,E2 27713.722} C_VEL
LIN {X 0,Y 585.241,Z 306.279,A -85,B 0,C 180,E1 27710.461,E2 27710.461} C_VEL
LIN {X 0,Y 585.253,Z 306.316,A -85,B 0,C 180,E1 27707.167,E2 27707.167} C_VEL
LIN {X 0,Y 585.25,Z 306.305,A -85,B 0,C 180,E1 27703.83,E2 27703.83} C_VEL
LIN {X 0,Y 585.233,Z 306.283,A -85,B 0,C 180,E1 27700.575,E2 27700.575} C_VEL
LIN {X 0,Y 585.25,Z 306.314,A -85,B 0,C 180,E1 27697.302,E2 27697.302} C_VEL
LIN {X 0,Y 585.242,Z 306.308,A -85,B 0,C 180,E1 27694.063,E2 27694.063} C_VEL
LIN {X 0,Y 585.289,Z 306.635,A -85,B 0,C 180,E1 27692.587,E2 27692.587} C_VEL
LIN {X 0,Y 586.744,Z 310.038,A -85,B 0,C 180,E1 27691.833,E2 27691.833} C_VEL
LIN {X 0,Y 588.391,Z 312.289,A -85,B 0,C 180,E1 27691.254,E2 27691.254} C_VEL
LIN {X 0,Y 590.357,Z 315.959,A -85,B 0,C 180,E1 27690.471,E2 27690.471} C_VEL
LIN {X 0,Y 591.453,Z 317.683,A -85,B 0,C 180,E1 27690.085,E2 27690.085} C_VEL
LIN {X 0,Y 593.586,Z 321.414,A -85,B 0,C 180,E1 27689.309,E2 27689.309} C_VEL
LIN {X 0,Y 597.356,Z 328.433,A -85,B 0,C 180,E1 27687.953,E2 27687.953} C_VEL
LIN {X 0,Y 602.288,Z 337.451,A -85,B 0,C 180,E1 27686.324,E2 27686.324} C_VEL
LIN {X 0,Y 608.671,Z 349.823,A -85,B 0,C 180,E1 27684.326,E2 27684.326} C_VEL
LIN {X 0,Y 620.381,Z 366.764,A -85,B 0,C 180,E1 27682.553,E2 27682.553} C_VEL
LIN {X 0,Y 631.477,Z 383.46,A -85,B 0,C 180,E1 27681.032,E2 27681.032} C_VEL
LIN {X 0,Y 633.595,Z 395.109,A -85,B 0,C 180,E1 27680.611,E2 27680.611} C_VEL
LIN {X 0,Y 628.489,Z 604.871,A -85,B 0,C 180,E1 27677.681,E2 27677.681} C_VEL
LIN {X 0,Y 623.606,Z 823.53,A -85,B 0,C 180,E1 27674.71,E2 27674.71} C_VEL
LIN {X 0,Y 622.568,Z 845.625,A -85,B 0,C 180,E1 27674.337,E2 27674.337} C_VEL
LIN {X 0,Y 621.166,Z 868.631,A -85,B 0,C 180,E1 27673.828,E2 27673.828} C_VEL
LIN {X 0,Y 619.047,Z 896.71,A -85,B 0,C 180,E1 27673.032,E2 27673.032} C_VEL
LIN {X 0,Y 617.041,Z 918.717,A -85,B 0,C 180,E1 27672.258,E2 27672.258} C_VEL
LIN {X 0,Y 614.817,Z 939.453,A -85,B 0,C 180,E1 27671.382,E2 27671.382} C_VEL
LIN {X 0,Y 612.607,Z 958.138,A -85,B 0,C 180,E1 27670.483,E2 27670.483} C_VEL
LIN {X 0,Y 610.25,Z 976.732,A -85,B 0,C 180,E1 27669.473,E2 27669.473} C_VEL
LIN {X 0,Y 607.667,Z 996.103,A -85,B 0,C 180,E1 27668.29,E2 27668.29} C_VEL
LIN {X 0,Y 604.564,Z 1018.85,A -85,B 0,C 180,E1 27666.717,E2 27666.717} C_VEL
LIN {X 0,Y 601.295,Z 1041.165,A -85,B 0,C 180,E1 27664.934,E2 27664.934} C_VEL
LIN {X 0,Y 598.8,Z 1058.371,A -85,B 0,C 180,E1 27663.393,E2 27663.393} C_VEL
LIN {X 0,Y 596.369,Z 1075.328,A -85,B 0,C 180,E1 27661.709,E2 27661.709} C_VEL
LIN {X 0,Y 593.58,Z 1095.644,A -85,B 0,C 180,E1 27659.437,E2 27659.437} C_VEL
LIN {X 0,Y 591.382,Z 1111.843,A -85,B 0,C 180,E1 27657.379,E2 27657.379} C_VEL
LIN {X 0,Y 589.581,Z 1126.359,A -85,B 0,C 180,E1 27655.32,E2 27655.32} C_VEL
LIN {X 0,Y 587.766,Z 1142.54,A -85,B 0,C 180,E1 27652.715,E2 27652.715} C_VEL
LIN {X 0,Y 586.534,Z 1154.754,A -85,B 0,C 180,E1 27650.454,E2 27650.454} C_VEL
LIN {X 0,Y 585.667,Z 1164.988,A -85,B 0,C 180,E1 27648.308,E2 27648.308} C_VEL
LIN {X 0,Y 584.904,Z 1175.544,A -85,B 0,C 180,E1 27645.772,E2 27645.772} C_VEL
LIN {X 0,Y 584.405,Z 1184.873,A -85,B 0,C 180,E1 27643.052,E2 27643.052} C_VEL
LIN {X 0,Y 584.13,Z 1191.439,A -85,B 0,C 180,E1 27640.718,E2 27640.718} C_VEL
LIN {X 0,Y 583.995,Z 1196.977,A -85,B 0,C 180,E1 27638.258,E2 27638.258} C_VEL
LIN {X 0,Y 583.93,Z 1201.428,A -85,B 0,C 180,E1 27635.503,E2 27635.503} C_VEL
LIN {X 0,Y 583.917,Z 1203.854,A -85,B 0,C 180,E1 27633.043,E2 27633.043} C_VEL
LIN {X 0,Y 583.905,Z 1204.804,A -85,B 0,C 180,E1 27630.883,E2 27630.883} C_VEL
LIN {X 0,Y 583.915,Z 1204.736,A -85,B 0,C 180,E1 27628.823,E2 27628.823} C_VEL
LIN {X 0,Y 583.913,Z 1203.51,A -85,B 0,C 180,E1 27626.466,E2 27626.466} C_VEL
LIN {X 0,Y 583.943,Z 1200.337,A -85,B 0,C 180,E1 27623.709,E2 27623.709} C_VEL
LIN {X 0,Y 584.019,Z 1195.926,A -85,B 0,C 180,E1 27621.236,E2 27621.236} C_VEL
LIN {X 0,Y 584.152,Z 1190.586,A -85,B 0,C 180,E1 27618.948,E2 27618.948} C_VEL
LIN {X 0,Y 584.519,Z 1182.685,A -85,B 0,C 180,E1 27616.245,E2 27616.245} C_VEL
LIN {X 0,Y 585.07,Z 1173.114,A -85,B 0,C 180,E1 27613.622,E2 27613.622} C_VEL
LIN {X 0,Y 585.743,Z 1164.074,A -85,B 0,C 180,E1 27611.488,E2 27611.488} C_VEL
LIN {X 0,Y 586.693,Z 1153.206,A -85,B 0,C 180,E1 27609.239,E2 27609.239} C_VEL
LIN {X 0,Y 588.226,Z 1138.277,A -85,B 0,C 180,E1 27606.563,E2 27606.563} C_VEL
LIN {X 0,Y 589.783,Z 1124.56,A -85,B 0,C 180,E1 27604.413,E2 27604.413} C_VEL
LIN {X 0,Y 591.601,Z 1110.303,A -85,B 0,C 180,E1 27602.414,E2 27602.414} C_VEL
LIN {X 0,Y 594.11,Z 1091.609,A -85,B 0,C 180,E1 27600.083,E2 27600.083} C_VEL
LIN {X 0,Y 596.592,Z 1073.81,A -85,B 0,C 180,E1 27598.135,E2 27598.135} C_VEL
LIN {X 0,Y 598.947,Z 1057.387,A -85,B 0,C 180,E1 27596.515,E2 27596.515} C_VEL
LIN {X 0,Y 601.698,Z 1038.571,A -85,B 0,C 180,E1 27594.845,E2 27594.845} C_VEL
LIN {X 0,Y 605.029,Z 1015.188,A -85,B 0,C 180,E1 27593.02,E2 27593.02} C_VEL
LIN {X 0,Y 607.749,Z 995.427,A -85,B 0,C 180,E1 27591.667,E2 27591.667} C_VEL
LIN {X 0,Y 610.362,Z 975.836,A -85,B 0,C 180,E1 27590.475,E2 27590.475} C_VEL
LIN {X 0,Y 612.906,Z 955.676,A -85,B 0,C 180,E1 27589.39,E2 27589.39} C_VEL
LIN {X 0,Y 615.754,Z 931.539,A -85,B 0,C 180,E1 27588.26,E2 27588.26} C_VEL
LIN {X 0,Y 618.108,Z 907.494,A -85,B 0,C 180,E1 27587.33,E2 27587.33} C_VEL
LIN {X 0,Y 619.978,Z 885.083,A -85,B 0,C 180,E1 27586.614,E2 27586.614} C_VEL
LIN {X 0,Y 621.539,Z 863.516,A -85,B 0,C 180,E1 27586.045,E2 27586.045} C_VEL
LIN {X 0,Y 622.833,Z 841.687,A -85,B 0,C 180,E1 27585.583,E2 27585.583} C_VEL
LIN {X 0,Y 624.015,Z 813.751,A -85,B 0,C 180,E1 27585.139,E2 27585.139} C_VEL
LIN {X 0,Y 628.981,Z 590.678,A -85,B 0,C 180,E1 27582.109,E2 27582.109} C_VEL
LIN {X 0,Y 633.767,Z 394.177,A -85,B 0,C 180,E1 27579.356,E2 27579.356} C_VEL
LIN {X 0,Y 631.352,Z 383.032,A -85,B 0,C 180,E1 27578.928,E2 27578.928} C_VEL
LIN {X 0,Y 612.096,Z 355.605,A -85,B 0,C 180,E1 27576.427,E2 27576.427} C_VEL
LIN {X 0,Y 607.469,Z 349.016,A -85,B 0,C 180,E1 27575.756,E2 27575.756} C_VEL
LIN {X 0,Y 597.539,Z 329.734,A -85,B 0,C 180,E1 27572.946,E2 27572.946} C_VEL
LIN {X 0,Y 592.074,Z 319.686,A -85,B 0,C 180,E1 27571.342,E2 27571.342} C_VEL
LIN {X 0,Y 589.949,Z 315.569,A -85,B 0,C 180,E1 27570.674,E2 27570.674} C_VEL
LIN {X 0,Y 587.164,Z 310.6,A -85,B 0,C 180,E1 27569.818,E2 27569.818} C_VEL
LIN {X 0,Y 585.402,Z 307.146,A -85,B 0,C 180,E1 27569.217,E2 27569.217} C_VEL
LIN {X 0,Y 585.262,Z 306.414,A -85,B 0,C 180,E1 27568.991,E2 27568.991} C_VEL
LIN {X 0,Y 585.238,Z 306.29,A -85,B 0,C 180,E1 27565.72,E2 27565.72} C_VEL
LIN {X 0,Y 585.238,Z 306.285,A -85,B 0,C 180,E1 27562.608,E2 27562.608} C_VEL
LIN {X 0,Y 585.246,Z 306.324,A -85,B 0,C 180,E1 27559.357,E2 27559.357} C_VEL
LIN {X 0,Y 585.248,Z 306.268,A -85,B 0,C 180,E1 27556.068,E2 27556.068} C_VEL
LIN {X 0,Y 585.25,Z 306.33,A -85,B 0,C 180,E1 27552.706,E2 27552.706} C_VEL
LIN {X 0,Y 585.241,Z 306.266,A -85,B 0,C 180,E1 27549.44,E2 27549.44} C_VEL
LIN {X 0,Y 585.237,Z 306.33,A -85,B 0,C 180,E1 27546.278,E2 27546.278} C_VEL
LIN {X 0,Y 585.25,Z 306.328,A -85,B 0,C 180,E1 27543.036,E2 27543.036} C_VEL
LIN {X 0,Y 585.24,Z 306.329,A -85,B 0,C 180,E1 27539.804,E2 27539.804} C_VEL
LIN {X 0,Y 585.248,Z 306.323,A -85,B 0,C 180,E1 27536.474,E2 27536.474} C_VEL
LIN {X 0,Y 585.257,Z 306.318,A -85,B 0,C 180,E1 27533.131,E2 27533.131} C_VEL
LIN {X 0,Y 585.227,Z 306.321,A -85,B 0,C 180,E1 27529.864,E2 27529.864} C_VEL
LIN {X 0,Y 585.254,Z 306.315,A -85,B 0,C 180,E1 27526.665,E2 27526.665} C_VEL
LIN {X 0,Y 585.226,Z 306.316,A -85,B 0,C 180,E1 27523.524,E2 27523.524} C_VEL
LIN {X 0,Y 585.252,Z 306.318,A -85,B 0,C 180,E1 27520.228,E2 27520.228} C_VEL
LIN {X 0,Y 585.248,Z 306.315,A -85,B 0,C 180,E1 27516.968,E2 27516.968} C_VEL
LIN {X 0,Y 585.219,Z 306.284,A -85,B 0,C 180,E1 27513.626,E2 27513.626} C_VEL
LIN {X 0,Y 585.259,Z 306.308,A -85,B 0,C 180,E1 27510.525,E2 27510.525} C_VEL
LIN {X 0,Y 585.211,Z 306.292,A -85,B 0,C 180,E1 27507.322,E2 27507.322} C_VEL
LIN {X 0,Y 585.256,Z 306.29,A -85,B 0,C 180,E1 27504.242,E2 27504.242} C_VEL
LIN {X 0,Y 585.21,Z 306.319,A -85,B 0,C 180,E1 27501.022,E2 27501.022} C_VEL
LIN {X 0,Y 585.248,Z 306.276,A -85,B 0,C 180,E1 27497.822,E2 27497.822} C_VEL
LIN {X 0,Y 585.25,Z 306.58,A -85,B 0,C 180,E1 27496.802,E2 27496.802} C_VEL
LIN {X 0,Y 586.63,Z 309.893,A -85,B 0,C 180,E1 27496.21,E2 27496.21} C_VEL
LIN {X 0,Y 587.703,Z 311.538,A -85,B 0,C 180,E1 27495.885,E2 27495.885} C_VEL
LIN {X 0,Y 589.484,Z 315.198,A -85,B 0,C 180,E1 27495.257,E2 27495.257} C_VEL
LIN {X 0,Y 594.604,Z 325.313,A -85,B 0,C 180,E1 27493.55,E2 27493.55} C_VEL
LIN {X 0,Y 602.623,Z 341.906,A -85,B 0,C 180,E1 27490.948,E2 27490.948} C_VEL
LIN {X 0,Y 605.399,Z 347.712,A -85,B 0,C 180,E1 27490.138,E2 27490.138} C_VEL
LIN {X 0,Y 621.714,Z 370.961,A -85,B 0,C 180,E1 27487.995,E2 27487.995} C_VEL
LIN {X 0,Y 625.717,Z 377.356,A -85,B 0,C 180,E1 27487.486,E2 27487.486} C_VEL
LIN {X 0,Y 628.355,Z 390.607,A -85,B 0,C 180,E1 27487.003,E2 27487.003} C_VEL
LIN {X 0,Y 627.068,Z 439.932,A -85,B 0,C 180,E1 27486.324,E2 27486.324} C_VEL
LIN {X 0,Y 626.185,Z 447.636,A -85,B 0,C 180,E1 27486.285,E2 27486.285} C_VEL
LIN {X 0,Y 621.341,Z 468.276,A -85,B 0,C 180,E1 27486.421,E2 27486.421} C_VEL
LIN {X 0,Y 620.646,Z 474.885,A -85,B 0,C 180,E1 27486.38,E2 27486.38} C_VEL
LIN {X 0,Y 614.605,Z 704.58,A -85,B 0,C 180,E1 27483.231,E2 27483.231} C_VEL
LIN {X 0,Y 612.396,Z 784.054,A -85,B 0,C 180,E1 27482.127,E2 27482.127} C_VEL
LIN {X 0,Y 610.873,Z 811.788,A -85,B 0,C 180,E1 27481.578,E2 27481.578} C_VEL
LIN {X 0,Y 609.249,Z 833.356,A -85,B 0,C 180,E1 27481.005,E2 27481.005} C_VEL
LIN {X 0,Y 607.401,Z 854.086,A -85,B 0,C 180,E1 27480.328,E2 27480.328} C_VEL
LIN {X 0,Y 604.889,Z 878.777,A -85,B 0,C 180,E1 27479.347,E2 27479.347} C_VEL
LIN {X 0,Y 602.368,Z 899.791,A -85,B 0,C 180,E1 27478.341,E2 27478.341} C_VEL
LIN {X 0,Y 600.014,Z 918.101,A -85,B 0,C 180,E1 27477.334,E2 27477.334} C_VEL
LIN {X 0,Y 597.368,Z 937.527,A -85,B 0,C 180,E1 27476.117,E2 27476.117} C_VEL
LIN {X 0,Y 594.048,Z 960.364,A -85,B 0,C 180,E1 27474.459,E2 27474.459} C_VEL
LIN {X 0,Y 591.384,Z 978.003,A -85,B 0,C 180,E1 27472.989,E2 27472.989} C_VEL
LIN {X 0,Y 588.69,Z 995.863,A -85,B 0,C 180,E1 27471.313,E2 27471.313} C_VEL
LIN {X 0,Y 585.58,Z 1016.994,A -85,B 0,C 180,E1 27469.034,E2 27469.034} C_VEL
LIN {X 0,Y 583.396,Z 1033.64,A -85,B 0,C 180,E1 27467.042,E2 27467.042} C_VEL
LIN {X 0,Y 581.409,Z 1049.634,A -85,B 0,C 180,E1 27464.847,E2 27464.847} C_VEL
LIN {X 0,Y 579.992,Z 1061.889,A -85,B 0,C 180,E1 27462.95,E2 27462.95} C_VEL
LIN {X 0,Y 578.671,Z 1075.057,A -85,B 0,C 180,E1 27460.654,E2 27460.654} C_VEL
LIN {X 0,Y 577.618,Z 1086.758,A -85,B 0,C 180,E1 27458.26,E2 27458.26} C_VEL
LIN {X 0,Y 576.971,Z 1095.615,A -85,B 0,C 180,E1 27456.168,E2 27456.168} C_VEL
LIN {X 0,Y 576.465,Z 1104.288,A -85,B 0,C 180,E1 27453.779,E2 27453.779} C_VEL
LIN {X 0,Y 576.157,Z 1111.529,A -85,B 0,C 180,E1 27451.293,E2 27451.293} C_VEL
LIN {X 0,Y 576.007,Z 1116.399,A -85,B 0,C 180,E1 27449.204,E2 27449.204} C_VEL
LIN {X 0,Y 575.939,Z 1120.18,A -85,B 0,C 180,E1 27447.114,E2 27447.114} C_VEL
LIN {X 0,Y 575.906,Z 1123.326,A -85,B 0,C 180,E1 27444.62,E2 27444.62} C_VEL
LIN {X 0,Y 575.917,Z 1124.743,A -85,B 0,C 180,E1 27442.117,E2 27442.117} C_VEL
LIN {X 0,Y 575.897,Z 1124.791,A -85,B 0,C 180,E1 27440.002,E2 27440.002} C_VEL
LIN {X 0,Y 575.912,Z 1123.698,A -85,B 0,C 180,E1 27437.817,E2 27437.817} C_VEL
LIN {X 0,Y 575.921,Z 1120.845,A -85,B 0,C 180,E1 27435.214,E2 27435.214} C_VEL
LIN {X 0,Y 575.994,Z 1116.882,A -85,B 0,C 180,E1 27432.94,E2 27432.94} C_VEL
LIN {X 0,Y 576.127,Z 1112.121,A -85,B 0,C 180,E1 27430.852,E2 27430.852} C_VEL
LIN {X 0,Y 576.381,Z 1105.864,A -85,B 0,C 180,E1 27428.636,E2 27428.636} C_VEL
LIN {X 0,Y 576.914,Z 1096.503,A -85,B 0,C 180,E1 27425.966,E2 27425.966} C_VEL
LIN {X 0,Y 577.535,Z 1087.932,A -85,B 0,C 180,E1 27423.913,E2 27423.913} C_VEL
LIN {X 0,Y 578.389,Z 1078.029,A -85,B 0,C 180,E1 27421.84,E2 27421.84} C_VEL
LIN {X 0,Y 579.792,Z 1064.006,A -85,B 0,C 180,E1 27419.306,E2 27419.306} C_VEL
LIN {X 0,Y 581.237,Z 1051.023,A -85,B 0,C 180,E1 27417.269,E2 27417.269} C_VEL
LIN {X 0,Y 583.098,Z 1036.041,A -85,B 0,C 180,E1 27415.18,E2 27415.18} C_VEL
LIN {X 0,Y 585.379,Z 1018.447,A -85,B 0,C 180,E1 27413.042,E2 27413.042} C_VEL
LIN {X 0,Y 588.603,Z 996.83,A -85,B 0,C 180,E1 27410.683,E2 27410.683} C_VEL
LIN {X 0,Y 591.387,Z 978.453,A -85,B 0,C 180,E1 27408.945,E2 27408.945} C_VEL
LIN {X 0,Y 594.156,Z 960.357,A -85,B 0,C 180,E1 27407.43,E2 27407.43} C_VEL
LIN {X 0,Y 597.435,Z 938.127,A -85,B 0,C 180,E1 27405.809,E2 27405.809} C_VEL
LIN {X 0,Y 600.124,Z 918.638,A -85,B 0,C 180,E1 27404.582,E2 27404.582} C_VEL
LIN {X 0,Y 602.648,Z 899.329,A -85,B 0,C 180,E1 27403.516,E2 27403.516} C_VEL
LIN {X 0,Y 605.486,Z 875.399,A -85,B 0,C 180,E1 27402.385,E2 27402.385} C_VEL
LIN {X 0,Y 607.793,Z 852.735,A -85,B 0,C 180,E1 27401.504,E2 27401.504} C_VEL
LIN {X 0,Y 609.703,Z 831.283,A -85,B 0,C 180,E1 27400.811,E2 27400.811} C_VEL
LIN {X 0,Y 611.635,Z 804.336,A -85,B 0,C 180,E1 27400.129,E2 27400.129} C_VEL
LIN {X 0,Y 612.834,Z 781.059,A -85,B 0,C 180,E1 27399.705,E2 27399.705} C_VEL
LIN {X 0,Y 619.533,Z 545.819,A -85,B 0,C 180,E1 27396.44,E2 27396.44} C_VEL
LIN {X 0,Y 624.092,Z 391.414,A -85,B 0,C 180,E1 27394.254,E2 27394.254} C_VEL
LIN {X 0,Y 622.169,Z 382.059,A -85,B 0,C 180,E1 27393.867,E2 27393.867} C_VEL
LIN {X 0,Y 611.255,Z 365.504,A -85,B 0,C 180,E1 27392.227,E2 27392.227} C_VEL
LIN {X 0,Y 599.6,Z 349.349,A -85,B 0,C 180,E1 27390.35,E2 27390.35} C_VEL
LIN {X 0,Y 597.616,Z 346.329,A -85,B 0,C 180,E1 27389.928,E2 27389.928} C_VEL
LIN {X 0,Y 592.199,Z 335.464,A -85,B 0,C 180,E1 27387.885,E2 27387.885} C_VEL
LIN {X 0,Y 587.57,Z 326.56,A -85,B 0,C 180,E1 27386.043,E2 27386.043} C_VEL
LIN {X 0,Y 584.977,Z 321.745,A -85,B 0,C 180,E1 27384.973,E2 27384.973} C_VEL
LIN {X 0,Y 582.486,Z 317.115,A -85,B 0,C 180,E1 27383.899,E2 27383.899} C_VEL
LIN {X 0,Y 580.464,Z 313.565,A -85,B 0,C 180,E1 27383.018,E2 27383.018} C_VEL
LIN {X 0,Y 579.599,Z 312.013,A -85,B 0,C 180,E1 27382.626,E2 27382.626} C_VEL
LIN {X 0,Y 577.51,Z 308.334,A -85,B 0,C 180,E1 27381.641,E2 27381.641} C_VEL
LIN {X 0,Y 577.324,Z 307.377,A -85,B 0,C 180,E1 27381.29,E2 27381.29} C_VEL
LIN {X 0,Y 577.311,Z 307.277,A -85,B 0,C 180,E1 27377.956,E2 27377.956} C_VEL
LIN {X 0,Y 577.308,Z 307.32,A -85,B 0,C 180,E1 27374.648,E2 27374.648} C_VEL
LIN {X 0,Y 577.303,Z 307.273,A -85,B 0,C 180,E1 27371.388,E2 27371.388} C_VEL
LIN {X 0,Y 577.298,Z 307.284,A -85,B 0,C 180,E1 27368.165,E2 27368.165} C_VEL
LIN {X 0,Y 577.305,Z 307.304,A -85,B 0,C 180,E1 27364.968,E2 27364.968} C_VEL
LIN {X 0,Y 577.307,Z 307.266,A -85,B 0,C 180,E1 27361.687,E2 27361.687} C_VEL
LIN {X 0,Y 577.315,Z 307.315,A -85,B 0,C 180,E1 27358.313,E2 27358.313} C_VEL
LIN {X 0,Y 577.3,Z 307.276,A -85,B 0,C 180,E1 27355.032,E2 27355.032} C_VEL
LIN {X 0,Y 577.302,Z 307.281,A -85,B 0,C 180,E1 27351.835,E2 27351.835} C_VEL
LIN {X 0,Y 577.301,Z 307.308,A -85,B 0,C 180,E1 27348.604,E2 27348.604} C_VEL
LIN {X 0,Y 577.308,Z 307.267,A -85,B 0,C 180,E1 27345.352,E2 27345.352} C_VEL
LIN {X 0,Y 577.314,Z 307.299,A -85,B 0,C 180,E1 27342.044,E2 27342.044} C_VEL
LIN {X 0,Y 577.3,Z 307.297,A -85,B 0,C 180,E1 27338.671,E2 27338.671} C_VEL
LIN {X 0,Y 577.306,Z 307.269,A -85,B 0,C 180,E1 27335.404,E2 27335.404} C_VEL
LIN {X 0,Y 577.347,Z 307.61,A -85,B 0,C 180,E1 27334.092,E2 27334.092} C_VEL
LIN {X 0,Y 578.959,Z 311.267,A -85,B 0,C 180,E1 27333.207,E2 27333.207} C_VEL
LIN {X 0,Y 580.524,Z 313.37,A -85,B 0,C 180,E1 27332.621,E2 27332.621} C_VEL
LIN {X 0,Y 582.376,Z 316.839,A -85,B 0,C 180,E1 27331.826,E2 27331.826} C_VEL
LIN {X 0,Y 583.475,Z 318.327,A -85,B 0,C 180,E1 27331.437,E2 27331.437} C_VEL
LIN {X 0,Y 585.821,Z 322.557,A -85,B 0,C 180,E1 27330.511,E2 27330.511} C_VEL
LIN {X 0,Y 589.524,Z 329.335,A -85,B 0,C 180,E1 27329.115,E2 27329.115} C_VEL
LIN {X 0,Y 592.602,Z 335.006,A -85,B 0,C 180,E1 27328.007,E2 27328.007} C_VEL
LIN {X 0,Y 597.221,Z 343.499,A -85,B 0,C 180,E1 27326.461,E2 27326.461} C_VEL
LIN {X 0,Y 600.805,Z 350.174,A -85,B 0,C 180,E1 27325.365,E2 27325.365} C_VEL
LIN {X 0,Y 611.36,Z 365.134,A -85,B 0,C 180,E1 27323.668,E2 27323.668} C_VEL
LIN {X 0,Y 626.682,Z 388.058,A -85,B 0,C 180,E1 27321.46,E2 27321.46} C_VEL
LIN {X 0,Y 628.261,Z 397.143,A -85,B 0,C 180,E1 27321.133,E2 27321.133} C_VEL
LIN {X 0,Y 622.9,Z 600.673,A -85,B 0,C 180,E1 27318.258,E2 27318.258} C_VEL
LIN {X 0,Y 617.719,Z 820.667,A -85,B 0,C 180,E1 27315.245,E2 27315.245} C_VEL
LIN {X 0,Y 616.636,Z 843.408,A -85,B 0,C 180,E1 27314.868,E2 27314.868} C_VEL
LIN {X 0,Y 615.274,Z 865.106,A -85,B 0,C 180,E1 27314.398,E2 27314.398} C_VEL
LIN {X 0,Y 613.462,Z 888.921,A -85,B 0,C 180,E1 27313.753,E2 27313.753} C_VEL
LIN {X 0,Y 610.859,Z 917.277,A -85,B 0,C 180,E1 27312.787,E2 27312.787} C_VEL
LIN {X 0,Y 608.668,Z 938.593,A -85,B 0,C 180,E1 27311.912,E2 27311.912} C_VEL
LIN {X 0,Y 606.685,Z 955.664,A -85,B 0,C 180,E1 27311.115,E2 27311.115} C_VEL
LIN {X 0,Y 604.011,Z 975.828,A -85,B 0,C 180,E1 27310.024,E2 27310.024} C_VEL
LIN {X 0,Y 601.263,Z 995.429,A -85,B 0,C 180,E1 27308.824,E2 27308.824} C_VEL
LIN {X 0,Y 598.199,Z 1016.662,A -85,B 0,C 180,E1 27307.354,E2 27307.354} C_VEL
LIN {X 0,Y 594.741,Z 1039.483,A -85,B 0,C 180,E1 27305.54,E2 27305.54} C_VEL
LIN {X 0,Y 591.985,Z 1057.385,A -85,B 0,C 180,E1 27303.932,E2 27303.932} C_VEL
LIN {X 0,Y 589.49,Z 1073.807,A -85,B 0,C 180,E1 27302.295,E2 27302.295} C_VEL
LIN {X 0,Y 586.83,Z 1091.626,A -85,B 0,C 180,E1 27300.324,E2 27300.324} C_VEL
LIN {X 0,Y 584.178,Z 1110.3,A -85,B 0,C 180,E1 27297.967,E2 27297.967} C_VEL
LIN {X 0,Y 582.255,Z 1124.381,A -85,B 0,C 180,E1 27295.969,E2 27295.969} C_VEL
LIN {X 0,Y 580.632,Z 1137.636,A -85,B 0,C 180,E1 27293.871,E2 27293.871} C_VEL
LIN {X 0,Y 578.983,Z 1152.68,A -85,B 0,C 180,E1 27291.157,E2 27291.157} C_VEL
LIN {X 0,Y 577.919,Z 1163.752,A -85,B 0,C 180,E1 27288.844,E2 27288.844} C_VEL
LIN {X 0,Y 577.173,Z 1172.908,A -85,B 0,C 180,E1 27286.661,E2 27286.661} C_VEL
LIN {X 0,Y 576.611,Z 1181.747,A -85,B 0,C 180,E1 27284.221,E2 27284.221} C_VEL
LIN {X 0,Y 576.219,Z 1189.82,A -85,B 0,C 180,E1 27281.511,E2 27281.511} C_VEL
LIN {X 0,Y 576.032,Z 1195.51,A -85,B 0,C 180,E1 27279.088,E2 27279.088} C_VEL
LIN {X 0,Y 575.948,Z 1199.726,A -85,B 0,C 180,E1 27276.763,E2 27276.763} C_VEL
LIN {X 0,Y 575.919,Z 1202.993,A -85,B 0,C 180,E1 27274.182,E2 27274.182} C_VEL
LIN {X 0,Y 575.908,Z 1204.646,A -85,B 0,C 180,E1 27271.592,E2 27271.592} C_VEL
LIN {X 0,Y 575.896,Z 1204.849,A -85,B 0,C 180,E1 27269.304,E2 27269.304} C_VEL
LIN {X 0,Y 575.915,Z 1203.987,A -85,B 0,C 180,E1 27267.114,E2 27267.114} C_VEL
LIN {X 0,Y 575.928,Z 1201.881,A -85,B 0,C 180,E1 27264.821,E2 27264.821} C_VEL
LIN {X 0,Y 575.975,Z 1198.251,A -85,B 0,C 180,E1 27262.319,E2 27262.319} C_VEL
LIN {X 0,Y 576.121,Z 1192.618,A -85,B 0,C 180,E1 27259.602,E2 27259.602} C_VEL
LIN {X 0,Y 576.386,Z 1186.006,A -85,B 0,C 180,E1 27257.146,E2 27257.146} C_VEL
LIN {X 0,Y 576.788,Z 1178.795,A -85,B 0,C 180,E1 27254.926,E2 27254.926} C_VEL
LIN {X 0,Y 577.447,Z 1169.448,A -85,B 0,C 180,E1 27252.465,E2 27252.465} C_VEL
LIN {X 0,Y 578.507,Z 1157.331,A -85,B 0,C 180,E1 27249.777,E2 27249.777} C_VEL
LIN {X 0,Y 579.671,Z 1146.003,A -85,B 0,C 180,E1 27247.592,E2 27247.592} C_VEL
LIN {X 0,Y 581.164,Z 1133.194,A -85,B 0,C 180,E1 27245.396,E2 27245.396} C_VEL
LIN {X 0,Y 583.409,Z 1115.694,A -85,B 0,C 180,E1 27242.768,E2 27242.768} C_VEL
LIN {X 0,Y 585.541,Z 1100.496,A -85,B 0,C 180,E1 27240.763,E2 27240.763} C_VEL
LIN {X 0,Y 587.89,Z 1084.523,A -85,B 0,C 180,E1 27238.867,E2 27238.867} C_VEL
LIN {X 0,Y 590.911,Z 1064.598,A -85,B 0,C 180,E1 27236.755,E2 27236.755} C_VEL
LIN {X 0,Y 593.915,Z 1044.652,A -85,B 0,C 180,E1 27234.906,E2 27234.906} C_VEL
LIN {X 0,Y 596.631,Z 1026.82,A -85,B 0,C 180,E1 27233.427,E2 27233.427} C_VEL
LIN {X 0,Y 599.476,Z 1007.838,A -85,B 0,C 180,E1 27232.015,E2 27232.015} C_VEL
LIN {X 0,Y 602.968,Z 983.931,A -85,B 0,C 180,E1 27230.45,E2 27230.45} C_VEL
LIN {X 0,Y 605.933,Z 961.702,A -85,B 0,C 180,E1 27229.198,E2 27229.198} C_VEL
LIN {X 0,Y 608.111,Z 943.661,A -85,B 0,C 180,E1 27228.312,E2 27228.312} C_VEL
LIN {X 0,Y 610.399,Z 922.093,A -85,B 0,C 180,E1 27227.397,E2 27227.397} C_VEL
LIN {X 0,Y 612.4,Z 901.422,A -85,B 0,C 180,E1 27226.643,E2 27226.643} C_VEL
LIN {X 0,Y 614.309,Z 879.156,A -85,B 0,C 180,E1 27225.957,E2 27225.957} C_VEL
LIN {X 0,Y 616.355,Z 850.464,A -85,B 0,C 180,E1 27225.259,E2 27225.259} C_VEL
LIN {X 0,Y 617.619,Z 825.864,A -85,B 0,C 180,E1 27224.822,E2 27224.822} C_VEL
LIN {X 0,Y 622.539,Z 623.424,A -85,B 0,C 180,E1 27222.04,E2 27222.04} C_VEL
LIN {X 0,Y 627.95,Z 412.061,A -85,B 0,C 180,E1 27219.071,E2 27219.071} C_VEL
LIN {X 0,Y 628.213,Z 395.631,A -85,B 0,C 180,E1 27218.823,E2 27218.823} C_VEL
LIN {X 0,Y 626.462,Z 387.791,A -85,B 0,C 180,E1 27218.512,E2 27218.512} C_VEL
LIN {X 0,Y 608.082,Z 361.575,A -85,B 0,C 180,E1 27216.092,E2 27216.092} C_VEL
LIN {X 0,Y 599.151,Z 348.958,A -85,B 0,C 180,E1 27214.802,E2 27214.802} C_VEL
LIN {X 0,Y 589.343,Z 330.229,A -85,B 0,C 180,E1 27211.961,E2 27211.961} C_VEL
LIN {X 0,Y 584.258,Z 320.805,A -85,B 0,C 180,E1 27210.401,E2 27210.401} C_VEL
LIN {X 0,Y 581.942,Z 316.486,A -85,B 0,C 180,E1 27209.659,E2 27209.659} C_VEL
LIN {X 0,Y 579.245,Z 311.611,A -85,B 0,C 180,E1 27208.791,E2 27208.791} C_VEL
LIN {X 0,Y 577.448,Z 308.053,A -85,B 0,C 180,E1 27208.155,E2 27208.155} C_VEL
LIN {X 0,Y 577.318,Z 307.391,A -85,B 0,C 180,E1 27207.961,E2 27207.961} C_VEL
LIN {X 0,Y 577.307,Z 307.308,A -85,B 0,C 180,E1 27204.781,E2 27204.781} C_VEL
LIN {X 0,Y 577.298,Z 307.261,A -85,B 0,C 180,E1 27201.542,E2 27201.542} C_VEL
LIN {X 0,Y 577.309,Z 307.315,A -85,B 0,C 180,E1 27198.27,E2 27198.27} C_VEL
LIN {X 0,Y 577.31,Z 307.265,A -85,B 0,C 180,E1 27194.853,E2 27194.853} C_VEL
LIN {X 0,Y 577.309,Z 307.293,A -85,B 0,C 180,E1 27191.59,E2 27191.59} C_VEL
LIN {X 0,Y 577.294,Z 307.269,A -85,B 0,C 180,E1 27188.366,E2 27188.366} C_VEL
LIN {X 0,Y 577.309,Z 307.308,A -85,B 0,C 180,E1 27185.167,E2 27185.167} C_VEL
LIN {X 0,Y 577.3,Z 307.311,A -85,B 0,C 180,E1 27181.886,E2 27181.886} C_VEL
LIN {X 0,Y 577.311,Z 307.31,A -85,B 0,C 180,E1 27178.511,E2 27178.511} C_VEL
LIN {X 0,Y 577.316,Z 307.317,A -85,B 0,C 180,E1 27175.231,E2 27175.231} C_VEL
LIN {X 0,Y 577.292,Z 307.321,A -85,B 0,C 180,E1 27172.035,E2 27172.035} C_VEL
LIN {X 0,Y 577.315,Z 307.315,A -85,B 0,C 180,E1 27168.815,E2 27168.815} C_VEL
LIN {X 0,Y 577.29,Z 307.319,A -85,B 0,C 180,E1 27165.557,E2 27165.557} C_VEL
LIN {X 0,Y 577.312,Z 307.31,A -85,B 0,C 180,E1 27162.252,E2 27162.252} C_VEL
LIN {X 0,Y 577.315,Z 307.309,A -85,B 0,C 180,E1 27158.987,E2 27158.987} C_VEL
LIN {X 0,Y 577.283,Z 307.268,A -85,B 0,C 180,E1 27155.764,E2 27155.764} C_VEL
LIN {X 0,Y 577.319,Z 307.303,A -85,B 0,C 180,E1 27152.568,E2 27152.568} C_VEL
LIN {X 0,Y 577.274,Z 307.269,A -85,B 0,C 180,E1 27149.387,E2 27149.387} C_VEL
LIN {X 0,Y 577.321,Z 307.314,A -85,B 0,C 180,E1 27146.104,E2 27146.104} C_VEL
LIN {X 0,Y 577.274,Z 307.264,A -85,B 0,C 180,E1 27142.931,E2 27142.931} C_VEL
LIN {X 0,Y 577.296,Z 307.296,A -85,B 0,C 180,E1 27139.626,E2 27139.626} C_VEL
LIN {X 0,Y 577.352,Z 307.541,A -85,B 0,C 180,E1 27137.858,E2 27137.858} C_VEL
LIN {X 0,Y 578.679,Z 310.91,A -85,B 0,C 180,E1 27137.23,E2 27137.23} C_VEL
LIN {X 0,Y 579.958,Z 313.054,A -85,B 0,C 180,E1 27136.807,E2 27136.807} C_VEL
LIN {X 0,Y 582.668,Z 318.493,A -85,B 0,C 180,E1 27135.831,E2 27135.831} C_VEL
LIN {X 0,Y 587.412,Z 327.728,A -85,B 0,C 180,E1 27134.223,E2 27134.223} C_VEL
LIN {X 0,Y 593.281,Z 339.789,A -85,B 0,C 180,E1 27132.255,E2 27132.255} C_VEL
LIN {X 0,Y 597.168,Z 347.68,A -85,B 0,C 180,E1 27131.071,E2 27131.071} C_VEL
LIN {X 0,Y 611.273,Z 367.766,A -85,B 0,C 180,E1 27129.145,E2 27129.145} C_VEL
LIN {X 0,Y 620.764,Z 381.791,A -85,B 0,C 180,E1 27127.911,E2 27127.911} C_VEL
LIN {X 0,Y 622.874,Z 392.655,A -85,B 0,C 180,E1 27127.518,E2 27127.518} C_VEL
LIN {X 0,Y 620.646,Z 474.885,A -85,B 0,C 180,E1 27126.38,E2 27126.38} C_VEL
LIN {X 0,Y 619.756,Z 482.587,A -85,B 0,C 180,E1 27126.341,E2 27126.341} C_VEL
LIN {X 0,Y 614.895,Z 503.216,A -85,B 0,C 180,E1 27126.48,E2 27126.48} C_VEL
LIN {X 0,Y 614.183,Z 509.825,A -85,B 0,C 180,E1 27126.441,E2 27126.441} C_VEL
LIN {X 0,Y 607.9,Z 741.769,A -85,B 0,C 180,E1 27123.249,E2 27123.249} C_VEL
LIN {X 0,Y 606.465,Z 788.153,A -85,B 0,C 180,E1 27122.584,E2 27122.584} C_VEL
LIN {X 0,Y 604.913,Z 813.59,A -85,B 0,C 180,E1 27122.058,E2 27122.058} C_VEL
LIN {X 0,Y 603.264,Z 834.57,A -85,B 0,C 180,E1 27121.493,E2 27121.493} C_VEL
LIN {X 0,Y 601.266,Z 856.064,A -85,B 0,C 180,E1 27120.781,E2 27120.781} C_VEL
LIN {X 0,Y 598.5,Z 881.459,A -85,B 0,C 180,E1 27119.747,E2 27119.747} C_VEL
LIN {X 0,Y 596.003,Z 901.318,A -85,B 0,C 180,E1 27118.782,E2 27118.782} C_VEL
LIN {X 0,Y 593.531,Z 919.603,A -85,B 0,C 180,E1 27117.761,E2 27117.761} C_VEL
LIN {X 0,Y 590.468,Z 941.119,A -85,B 0,C 180,E1 27116.388,E2 27116.388} C_VEL
LIN {X 0,Y 587.198,Z 962.104,A -85,B 0,C 180,E1 27114.823,E2 27114.823} C_VEL
LIN {X 0,Y 584.496,Z 979.146,A -85,B 0,C 180,E1 27113.382,E2 27113.382} C_VEL
LIN {X 0,Y 581.508,Z 997.979,A -85,B 0,C 180,E1 27111.59,E2 27111.59} C_VEL
LIN {X 0,Y 578.594,Z 1016.134,A -85,B 0,C 180,E1 27109.588,E2 27109.588} C_VEL
LIN {X 0,Y 576.122,Z 1032.335,A -85,B 0,C 180,E1 27107.576,E2 27107.576} C_VEL
LIN {X 0,Y 573.879,Z 1049.167,A -85,B 0,C 180,E1 27105.253,E2 27105.253} C_VEL
LIN {X 0,Y 572.282,Z 1062.074,A -85,B 0,C 180,E1 27103.231,E2 27103.231} C_VEL
LIN {X 0,Y 570.874,Z 1075.222,A -85,B 0,C 180,E1 27100.903,E2 27100.903} C_VEL
LIN {X 0,Y 569.746,Z 1086.888,A -85,B 0,C 180,E1 27098.477,E2 27098.477} C_VEL
LIN {X 0,Y 569.044,Z 1095.729,A -85,B 0,C 180,E1 27096.355,E2 27096.355} C_VEL
LIN {X 0,Y 568.491,Z 1104.725,A -85,B 0,C 180,E1 27093.832,E2 27093.832} C_VEL
LIN {X 0,Y 568.166,Z 1111.849,A -85,B 0,C 180,E1 27091.311,E2 27091.311} C_VEL
LIN {X 0,Y 568.01,Z 1116.66,A -85,B 0,C 180,E1 27089.193,E2 27089.193} C_VEL
LIN {X 0,Y 567.936,Z 1120.541,A -85,B 0,C 180,E1 27086.972,E2 27086.972} C_VEL
LIN {X 0,Y 567.899,Z 1123.558,A -85,B 0,C 180,E1 27084.342,E2 27084.342} C_VEL
LIN {X 0,Y 567.917,Z 1124.748,A -85,B 0,C 180,E1 27082.107,E2 27082.107} C_VEL
LIN {X 0,Y 567.896,Z 1124.807,A -85,B 0,C 180,E1 27080.064,E2 27080.064} C_VEL
LIN {X 0,Y 567.911,Z 1123.787,A -85,B 0,C 180,E1 27077.906,E2 27077.906} C_VEL
LIN {X 0,Y 567.93,Z 1121.285,A -85,B 0,C 180,E1 27075.419,E2 27075.419} C_VEL
LIN {X 0,Y 567.997,Z 1117.038,A -85,B 0,C 180,E1 27072.904,E2 27072.904} C_VEL
LIN {X 0,Y 568.14,Z 1112.313,A -85,B 0,C 180,E1 27070.786,E2 27070.786} C_VEL
LIN {X 0,Y 568.409,Z 1106.051,A -85,B 0,C 180,E1 27068.524,E2 27068.524} C_VEL
LIN {X 0,Y 568.986,Z 1096.654,A -85,B 0,C 180,E1 27065.791,E2 27065.791} C_VEL
LIN {X 0,Y 569.675,Z 1087.787,A -85,B 0,C 180,E1 27063.637,E2 27063.637} C_VEL
LIN {X 0,Y 570.661,Z 1077.316,A -85,B 0,C 180,E1 27061.424,E2 27061.424} C_VEL
LIN {X 0,Y 572.138,Z 1063.46,A -85,B 0,C 180,E1 27058.909,E2 27058.909} C_VEL
LIN {X 0,Y 573.637,Z 1051.026,A -85,B 0,C 180,E1 27056.937,E2 27056.937} C_VEL
LIN {X 0,Y 575.524,Z 1036.612,A -85,B 0,C 180,E1 27054.897,E2 27054.897} C_VEL
LIN {X 0,Y 578.343,Z 1017.882,A -85,B 0,C 180,E1 27052.52,E2 27052.52} C_VEL
LIN {X 0,Y 580.845,Z 1002.378,A -85,B 0,C 180,E1 27050.773,E2 27050.773} C_VEL
LIN {X 0,Y 584.117,Z 982.176,A -85,B 0,C 180,E1 27048.775,E2 27048.775} C_VEL
LIN {X 0,Y 586.977,Z 964.339,A -85,B 0,C 180,E1 27047.239,E2 27047.239} C_VEL
LIN {X 0,Y 589.955,Z 945.486,A -85,B 0,C 180,E1 27045.802,E2 27045.802} C_VEL
LIN {X 0,Y 593.419,Z 922.163,A -85,B 0,C 180,E1 27044.268,E2 27044.268} C_VEL
LIN {X 0,Y 596.028,Z 903.201,A -85,B 0,C 180,E1 27043.193,E2 27043.193} C_VEL
LIN {X 0,Y 598.447,Z 884.267,A -85,B 0,C 180,E1 27042.256,E2 27042.256} C_VEL
LIN {X 0,Y 601.197,Z 860.704,A -85,B 0,C 180,E1 27041.26,E2 27041.26} C_VEL
LIN {X 0,Y 603.496,Z 836.366,A -85,B 0,C 180,E1 27040.431,E2 27040.431} C_VEL
LIN {X 0,Y 605.131,Z 816.242,A -85,B 0,C 180,E1 27039.875,E2 27039.875} C_VEL
LIN {X 0,Y 606.482,Z 795.751,A -85,B 0,C 180,E1 27039.425,E2 27039.425} C_VEL
LIN {X 0,Y 607.784,Z 764.313,A -85,B 0,C 180,E1 27038.923,E2 27038.923} C_VEL
LIN {X 0,Y 614.911,Z 524.864,A -85,B 0,C 180,E1 27035.581,E2 27035.581} C_VEL
LIN {X 0,Y 618.993,Z 393.413,A -85,B 0,C 180,E1 27033.702,E2 27033.702} C_VEL
LIN {X 0,Y 617.636,Z 386.982,A -85,B 0,C 180,E1 27033.424,E2 27033.424} C_VEL
LIN {X 0,Y 607.403,Z 371.312,A -85,B 0,C 180,E1 27031.844,E2 27031.844} C_VEL
LIN {X 0,Y 596.246,Z 355.723,A -85,B 0,C 180,E1 27030.011,E2 27030.011} C_VEL
LIN {X 0,Y 589.995,Z 347.235,A -85,B 0,C 180,E1 27028.882,E2 27028.882} C_VEL
LIN {X 0,Y 584.447,Z 336.504,A -85,B 0,C 180,E1 27026.741,E2 27026.741} C_VEL
LIN {X 0,Y 581.809,Z 331.536,A -85,B 0,C 180,E1 27025.664,E2 27025.664} C_VEL
LIN {X 0,Y 580.011,Z 327.939,A -85,B 0,C 180,E1 27024.875,E2 27024.875} C_VEL
LIN {X 0,Y 577.264,Z 322.995,A -85,B 0,C 180,E1 27023.694,E2 27023.694} C_VEL
LIN {X 0,Y 574.647,Z 318.192,A -85,B 0,C 180,E1 27022.495,E2 27022.495} C_VEL
LIN {X 0,Y 572.561,Z 314.523,A -85,B 0,C 180,E1 27021.514,E2 27021.514} C_VEL
LIN {X 0,Y 571.511,Z 312.787,A -85,B 0,C 180,E1 27021.018,E2 27021.018} C_VEL
LIN {X 0,Y 569.681,Z 309.705,A -85,B 0,C 180,E1 27020.118,E2 27020.118} C_VEL
LIN {X 0,Y 569.39,Z 308.433,A -85,B 0,C 180,E1 27019.704,E2 27019.704} C_VEL
LIN {X 0,Y 569.357,Z 308.26,A -85,B 0,C 180,E1 27016.424,E2 27016.424} C_VEL
LIN {X 0,Y 569.367,Z 308.267,A -85,B 0,C 180,E1 27013.197,E2 27013.197} C_VEL
LIN {X 0,Y 569.377,Z 308.305,A -85,B 0,C 180,E1 27009.808,E2 27009.808} C_VEL
LIN {X 0,Y 569.365,Z 308.254,A -85,B 0,C 180,E1 27006.453,E2 27006.453} C_VEL
LIN {X 0,Y 569.364,Z 308.284,A -85,B 0,C 180,E1 27003.222,E2 27003.222} C_VEL
LIN {X 0,Y 569.364,Z 308.28,A -85,B 0,C 180,E1 26999.899,E2 26999.899} C_VEL
LIN {X 0,Y 569.363,Z 308.256,A -85,B 0,C 180,E1 26996.678,E2 26996.678} C_VEL
LIN {X 0,Y 569.379,Z 308.308,A -85,B 0,C 180,E1 26993.243,E2 26993.243} C_VEL
LIN {X 0,Y 569.365,Z 308.257,A -85,B 0,C 180,E1 26989.885,E2 26989.885} C_VEL
LIN {X 0,Y 569.358,Z 308.273,A -85,B 0,C 180,E1 26986.627,E2 26986.627} C_VEL
LIN {X 0,Y 569.372,Z 308.295,A -85,B 0,C 180,E1 26983.366,E2 26983.366} C_VEL
LIN {X 0,Y 569.372,Z 308.255,A -85,B 0,C 180,E1 26979.967,E2 26979.967} C_VEL
LIN {X 0,Y 569.363,Z 308.27,A -85,B 0,C 180,E1 26976.699,E2 26976.699} C_VEL
LIN {X 0,Y 569.42,Z 308.579,A -85,B 0,C 180,E1 26975.739,E2 26975.739} C_VEL
LIN {X 0,Y 570.928,Z 312.105,A -85,B 0,C 180,E1 26974.813,E2 26974.813} C_VEL
LIN {X 0,Y 572.658,Z 314.363,A -85,B 0,C 180,E1 26974.118,E2 26974.118} C_VEL
LIN {X 0,Y 574.626,Z 318.059,A -85,B 0,C 180,E1 26973.205,E2 26973.205} C_VEL
LIN {X 0,Y 575.746,Z 319.66,A -85,B 0,C 180,E1 26972.767,E2 26972.767} C_VEL
LIN {X 0,Y 578.018,Z 323.619,A -85,B 0,C 180,E1 26971.819,E2 26971.819} C_VEL
LIN {X 0,Y 581.775,Z 330.312,A -85,B 0,C 180,E1 26970.331,E2 26970.331} C_VEL
LIN {X 0,Y 584.879,Z 336.088,A -85,B 0,C 180,E1 26969.145,E2 26969.145} C_VEL
LIN {X 0,Y 587.812,Z 341.467,A -85,B 0,C 180,E1 26968.08,E2 26968.08} C_VEL
LIN {X 0,Y 592.436,Z 349.92,A -85,B 0,C 180,E1 26966.56,E2 26966.56} C_VEL
LIN {X 0,Y 602.8,Z 364.09,A -85,B 0,C 180,E1 26964.801,E2 26964.801} C_VEL
LIN {X 0,Y 613.525,Z 379.954,A -85,B 0,C 180,E1 26963.119,E2 26963.119} C_VEL
LIN {X 0,Y 622.04,Z 393.198,A -85,B 0,C 180,E1 26961.876,E2 26961.876} C_VEL
LIN {X 0,Y 622.983,Z 399.28,A -85,B 0,C 180,E1 26961.662,E2 26961.662} C_VEL
LIN {X 0,Y 617.101,Z 607.231,A -85,B 0,C 180,E1 26958.696,E2 26958.696} C_VEL
LIN {X 0,Y 611.681,Z 822.896,A -85,B 0,C 180,E1 26955.713,E2 26955.713} C_VEL
LIN {X 0,Y 610.531,Z 845.083,A -85,B 0,C 180,E1 26955.334,E2 26955.334} C_VEL
LIN {X 0,Y 608.892,Z 869.498,A -85,B 0,C 180,E1 26954.786,E2 26954.786} C_VEL
LIN {X 0,Y 606.54,Z 897.138,A -85,B 0,C 180,E1 26953.981,E2 26953.981} C_VEL
LIN {X 0,Y 604.286,Z 919.736,A -85,B 0,C 180,E1 26953.171,E2 26953.171} C_VEL
LIN {X 0,Y 602.103,Z 939.847,A -85,B 0,C 180,E1 26952.328,E2 26952.328} C_VEL
LIN {X 0,Y 599.73,Z 959.587,A -85,B 0,C 180,E1 26951.387,E2 26951.387} C_VEL
LIN {X 0,Y 597.009,Z 980.871,A -85,B 0,C 180,E1 26950.233,E2 26950.233} C_VEL
LIN {X 0,Y 593.327,Z 1005.639,A -85,B 0,C 180,E1 26948.635,E2 26948.635} C_VEL
LIN {X 0,Y 590.18,Z 1025.555,A -85,B 0,C 180,E1 26947.155,E2 26947.155} C_VEL
LIN {X 0,Y 587.382,Z 1042.969,A -85,B 0,C 180,E1 26945.709,E2 26945.709} C_VEL
LIN {X 0,Y 584.6,Z 1060.166,A -85,B 0,C 180,E1 26944.123,E2 26944.123} C_VEL
LIN {X 0,Y 581.464,Z 1079.873,A -85,B 0,C 180,E1 26942.096,E2 26942.096} C_VEL
LIN {X 0,Y 578.615,Z 1097.985,A -85,B 0,C 180,E1 26939.96,E2 26939.96} C_VEL
LIN {X 0,Y 576.365,Z 1112.966,A -85,B 0,C 180,E1 26937.99,E2 26937.99} C_VEL
LIN {X 0,Y 574.254,Z 1127.881,A -85,B 0,C 180,E1 26935.803,E2 26935.803} C_VEL
LIN {X 0,Y 572.236,Z 1143.703,A -85,B 0,C 180,E1 26933.15,E2 26933.15} C_VEL
LIN {X 0,Y 570.921,Z 1155.265,A -85,B 0,C 180,E1 26930.932,E2 26930.932} C_VEL
LIN {X 0,Y 569.924,Z 1165.444,A -85,B 0,C 180,E1 26928.726,E2 26928.726} C_VEL
LIN {X 0,Y 569.029,Z 1176.303,A -85,B 0,C 180,E1 26926.016,E2 26926.016} C_VEL
LIN {X 0,Y 568.479,Z 1185.17,A -85,B 0,C 180,E1 26923.321,E2 26923.321} C_VEL
LIN {X 0,Y 568.16,Z 1191.597,A -85,B 0,C 180,E1 26920.956,E2 26920.956} C_VEL
LIN {X 0,Y 568.007,Z 1197.191,A -85,B 0,C 180,E1 26918.381,E2 26918.381} C_VEL
LIN {X 0,Y 567.932,Z 1201.538,A -85,B 0,C 180,E1 26915.557,E2 26915.557} C_VEL
LIN {X 0,Y 567.917,Z 1203.848,A -85,B 0,C 180,E1 26913.129,E2 26913.129} C_VEL
LIN {X 0,Y 567.906,Z 1204.804,A -85,B 0,C 180,E1 26910.908,E2 26910.908} C_VEL
LIN {X 0,Y 567.916,Z 1204.736,A -85,B 0,C 180,E1 26908.789,E2 26908.789} C_VEL
LIN {X 0,Y 567.912,Z 1203.507,A -85,B 0,C 180,E1 26906.366,E2 26906.366} C_VEL
LIN {X 0,Y 567.948,Z 1200.336,A -85,B 0,C 180,E1 26903.531,E2 26903.531} C_VEL
LIN {X 0,Y 568.029,Z 1196.127,A -85,B 0,C 180,E1 26901.089,E2 26901.089} C_VEL
LIN {X 0,Y 568.191,Z 1190.834,A -85,B 0,C 180,E1 26898.736,E2 26898.736} C_VEL
LIN {X 0,Y 568.577,Z 1183.471,A -85,B 0,C 180,E1 26896.107,E2 26896.107} C_VEL
LIN {X 0,Y 569.205,Z 1173.921,A -85,B 0,C 180,E1 26893.362,E2 26893.362} C_VEL
LIN {X 0,Y 570.006,Z 1164.53,A -85,B 0,C 180,E1 26891.064,E2 26891.064} C_VEL
LIN {X 0,Y 571.043,Z 1154.241,A -85,B 0,C 180,E1 26888.857,E2 26888.857} C_VEL
LIN {X 0,Y 572.616,Z 1140.801,A -85,B 0,C 180,E1 26886.321,E2 26886.321} C_VEL
LIN {X 0,Y 574.531,Z 1125.782,A -85,B 0,C 180,E1 26883.877,E2 26883.877} C_VEL
LIN {X 0,Y 576.537,Z 1111.839,A -85,B 0,C 180,E1 26881.854,E2 26881.854} C_VEL
LIN {X 0,Y 579.026,Z 1095.326,A -85,B 0,C 180,E1 26879.704,E2 26879.704} C_VEL
LIN {X 0,Y 582.167,Z 1075.371,A -85,B 0,C 180,E1 26877.428,E2 26877.428} C_VEL
LIN {X 0,Y 584.781,Z 1059.05,A -85,B 0,C 180,E1 26875.77,E2 26875.77} C_VEL
LIN {X 0,Y 587.479,Z 1042.377,A -85,B 0,C 180,E1 26874.24,E2 26874.24} C_VEL
LIN {X 0,Y 590.375,Z 1024.364,A -85,B 0,C 180,E1 26872.752,E2 26872.752} C_VEL
LIN {X 0,Y 594.048,Z 1001.028,A -85,B 0,C 180,E1 26871.044,E2 26871.044} C_VEL
LIN {X 0,Y 597.086,Z 980.246,A -85,B 0,C 180,E1 26869.731,E2 26869.731} C_VEL
LIN {X 0,Y 599.755,Z 959.616,A -85,B 0,C 180,E1 26868.61,E2 26868.61} C_VEL
LIN {X 0,Y 602.129,Z 940.065,A -85,B 0,C 180,E1 26867.674,E2 26867.674} C_VEL
LIN {X 0,Y 604.325,Z 920.076,A -85,B 0,C 180,E1 26866.832,E2 26866.832} C_VEL
LIN {X 0,Y 606.668,Z 896.881,A -85,B 0,C 180,E1 26865.998,E2 26865.998} C_VEL
LIN {X 0,Y 609.108,Z 868.116,A -85,B 0,C 180,E1 26865.167,E2 26865.167} C_VEL
LIN {X 0,Y 610.683,Z 844.841,A -85,B 0,C 180,E1 26864.647,E2 26864.647} C_VEL
LIN {X 0,Y 611.827,Z 822.782,A -85,B 0,C 180,E1 26864.27,E2 26864.27} C_VEL
LIN {X 0,Y 617.401,Z 604.669,A -85,B 0,C 180,E1 26861.247,E2 26861.247} C_VEL
LIN {X 0,Y 622.948,Z 398.35,A -85,B 0,C 180,E1 26858.329,E2 26858.329} C_VEL
LIN {X 0,Y 621.61,Z 392.511,A -85,B 0,C 180,E1 26858.089,E2 26858.089} C_VEL
LIN {X 0,Y 603.663,Z 366.97,A -85,B 0,C 180,E1 26855.694,E2 26855.694} C_VEL
LIN {X 0,Y 590.835,Z 349.084,A -85,B 0,C 180,E1 26853.833,E2 26853.833} C_VEL
LIN {X 0,Y 581.929,Z 331.905,A -85,B 0,C 180,E1 26851.144,E2 26851.144} C_VEL
LIN {X 0,Y 576.727,Z 322.356,A -85,B 0,C 180,E1 26849.497,E2 26849.497} C_VEL
LIN {X 0,Y 573.978,Z 317.419,A -85,B 0,C 180,E1 26848.603,E2 26848.603} C_VEL
LIN {X 0,Y 571.787,Z 313.125,A -85,B 0,C 180,E1 26847.834,E2 26847.834} C_VEL
LIN {X 0,Y 569.915,Z 310.315,A -85,B 0,C 180,E1 26847.253,E2 26847.253} C_VEL
LIN {X 0,Y 569.393,Z 308.453,A -85,B 0,C 180,E1 26846.903,E2 26846.903} C_VEL
LIN {X 0,Y 569.362,Z 308.288,A -85,B 0,C 180,E1 26843.604,E2 26843.604} C_VEL
LIN {X 0,Y 569.366,Z 308.265,A -85,B 0,C 180,E1 26840.348,E2 26840.348} C_VEL
LIN {X 0,Y 569.37,Z 308.255,A -85,B 0,C 180,E1 26837.054,E2 26837.054} C_VEL
LIN {X 0,Y 569.377,Z 308.29,A -85,B 0,C 180,E1 26833.714,E2 26833.714} C_VEL
LIN {X 0,Y 569.355,Z 308.246,A -85,B 0,C 180,E1 26830.421,E2 26830.421} C_VEL
LIN {X 0,Y 569.368,Z 308.294,A -85,B 0,C 180,E1 26827.163,E2 26827.163} C_VEL
LIN {X 0,Y 569.362,Z 308.297,A -85,B 0,C 180,E1 26823.927,E2 26823.927} C_VEL
LIN {X 0,Y 569.37,Z 308.295,A -85,B 0,C 180,E1 26820.503,E2 26820.503} C_VEL
LIN {X 0,Y 569.374,Z 308.289,A -85,B 0,C 180,E1 26817.182,E2 26817.182} C_VEL
LIN {X 0,Y 569.351,Z 308.293,A -85,B 0,C 180,E1 26813.951,E2 26813.951} C_VEL
LIN {X 0,Y 569.376,Z 308.294,A -85,B 0,C 180,E1 26810.702,E2 26810.702} C_VEL
LIN {X 0,Y 569.361,Z 308.299,A -85,B 0,C 180,E1 26807.422,E2 26807.422} C_VEL
LIN {X 0,Y 569.356,Z 308.297,A -85,B 0,C 180,E1 26803.995,E2 26803.995} C_VEL
LIN {X 0,Y 569.38,Z 308.301,A -85,B 0,C 180,E1 26800.722,E2 26800.722} C_VEL
LIN {X 0,Y 569.345,Z 308.306,A -85,B 0,C 180,E1 26797.478,E2 26797.478} C_VEL
LIN {X 0,Y 569.37,Z 308.243,A -85,B 0,C 180,E1 26794.181,E2 26794.181} C_VEL
LIN {X 0,Y 569.355,Z 308.303,A -85,B 0,C 180,E1 26790.991,E2 26790.991} C_VEL
LIN {X 0,Y 569.343,Z 308.256,A -85,B 0,C 180,E1 26787.612,E2 26787.612} C_VEL
LIN {X 0,Y 569.373,Z 308.27,A -85,B 0,C 180,E1 26784.459,E2 26784.459} C_VEL
LIN {X 0,Y 569.333,Z 308.285,A -85,B 0,C 180,E1 26781.172,E2 26781.172} C_VEL
LIN {X 0,Y 569.373,Z 308.562,A -85,B 0,C 180,E1 26778.944,E2 26778.944} C_VEL
LIN {X 0,Y 570.955,Z 312.114,A -85,B 0,C 180,E1 26778.246,E2 26778.246} C_VEL
LIN {X 0,Y 572.099,Z 314.094,A -85,B 0,C 180,E1 26777.845,E2 26777.845} C_VEL
LIN {X 0,Y 577.153,Z 324.046,A -85,B 0,C 180,E1 26775.995,E2 26775.995} C_VEL
LIN {X 0,Y 581.869,Z 333.308,A -85,B 0,C 180,E1 26774.368,E2 26774.368} C_VEL
LIN {X 0,Y 587.945,Z 345.982,A -85,B 0,C 180,E1 26772.287,E2 26772.287} C_VEL
LIN {X 0,Y 590.016,Z 349.341,A -85,B 0,C 180,E1 26771.875,E2 26771.875} C_VEL
LIN {X 0,Y 606.126,Z 371.993,A -85,B 0,C 180,E1 26769.63,E2 26769.63} C_VEL
LIN {X 0,Y 615.969,Z 386.745,A -85,B 0,C 180,E1 26768.321,E2 26768.321} C_VEL
LIN {X 0,Y 617.411,Z 394.648,A -85,B 0,C 180,E1 26768.039,E2 26768.039} C_VEL
LIN {X 0,Y 614.183,Z 509.825,A -85,B 0,C 180,E1 26766.441,E2 26766.441} C_VEL
LIN {X 0,Y 613.27,Z 517.53,A -85,B 0,C 180,E1 26766.404,E2 26766.404} C_VEL
LIN {X 0,Y 608.397,Z 538.158,A -85,B 0,C 180,E1 26766.544,E2 26766.544} C_VEL
LIN {X 0,Y 607.703,Z 544.765,A -85,B 0,C 180,E1 26766.503,E2 26766.503} C_VEL
LIN {X 0,Y 601.11,Z 777.425,A -85,B 0,C 180,E1 26763.281,E2 26763.281} C_VEL
LIN {X 0,Y 600.006,Z 799.691,A -85,B 0,C 180,E1 26762.893,E2 26762.893} C_VEL
LIN {X 0,Y 598.647,Z 819.736,A -85,B 0,C 180,E1 26762.435,E2 26762.435} C_VEL
LIN {X 0,Y 596.583,Z 844.305,A -85,B 0,C 180,E1 26761.725,E2 26761.725} C_VEL
LIN {X 0,Y 594.097,Z 867.596,A -85,B 0,C 180,E1 26760.867,E2 26760.867} C_VEL
LIN {X 0,Y 591.872,Z 886.204,A -85,B 0,C 180,E1 26760.058,E2 26760.058} C_VEL
LIN {X 0,Y 589.365,Z 905.209,A -85,B 0,C 180,E1 26759.105,E2 26759.105} C_VEL
LIN {X 0,Y 586.189,Z 927.553,A -85,B 0,C 180,E1 26757.808,E2 26757.808} C_VEL
LIN {X 0,Y 582.862,Z 948.493,A -85,B 0,C 180,E1 26756.378,E2 26756.378} C_VEL
LIN {X 0,Y 579.939,Z 966.43,A -85,B 0,C 180,E1 26754.986,E2 26754.986} C_VEL
LIN {X 0,Y 576.547,Z 986.871,A -85,B 0,C 180,E1 26753.183,E2 26753.183} C_VEL
LIN {X 0,Y 573.512,Z 1004.651,A -85,B 0,C 180,E1 26751.369,E2 26751.369} C_VEL
LIN {X 0,Y 570.991,Z 1019.697,A -85,B 0,C 180,E1 26749.646,E2 26749.646} C_VEL
LIN {X 0,Y 568.185,Z 1036.972,A -85,B 0,C 180,E1 26747.407,E2 26747.407} C_VEL
LIN {X 0,Y 565.465,Z 1055.427,A -85,B 0,C 180,E1 26744.646,E2 26744.646} C_VEL
LIN {X 0,Y 563.68,Z 1069.853,A -85,B 0,C 180,E1 26742.186,E2 26742.186} C_VEL
LIN {X 0,Y 562.519,Z 1080.393,A -85,B 0,C 180,E1 26740.135,E2 26740.135} C_VEL
LIN {X 0,Y 561.497,Z 1091.473,A -85,B 0,C 180,E1 26737.675,E2 26737.675} C_VEL
LIN {X 0,Y 560.764,Z 1101.028,A -85,B 0,C 180,E1 26735.115,E2 26735.115} C_VEL
LIN {X 0,Y 560.374,Z 1107.795,A -85,B 0,C 180,E1 26732.966,E2 26732.966} C_VEL
LIN {X 0,Y 560.093,Z 1114.177,A -85,B 0,C 180,E1 26730.511,E2 26730.511} C_VEL
LIN {X 0,Y 559.965,Z 1119.307,A -85,B 0,C 180,E1 26727.851,E2 26727.851} C_VEL
LIN {X 0,Y 559.911,Z 1122.253,A -85,B 0,C 180,E1 26725.699,E2 26725.699} C_VEL
LIN {X 0,Y 559.911,Z 1124.123,A -85,B 0,C 180,E1 26723.54,E2 26723.54} C_VEL
LIN {X 0,Y 559.909,Z 1124.983,A -85,B 0,C 180,E1 26721.062,E2 26721.062} C_VEL
LIN {X 0,Y 559.911,Z 1124.186,A -85,B 0,C 180,E1 26718.463,E2 26718.463} C_VEL
LIN {X 0,Y 559.912,Z 1122.426,A -85,B 0,C 180,E1 26716.366,E2 26716.366} C_VEL
LIN {X 0,Y 559.953,Z 1119.608,A -85,B 0,C 180,E1 26714.252,E2 26714.252} C_VEL
LIN {X 0,Y 560.064,Z 1115.268,A -85,B 0,C 180,E1 26711.902,E2 26711.902} C_VEL
LIN {X 0,Y 560.323,Z 1108.54,A -85,B 0,C 180,E1 26709.2,E2 26709.2} C_VEL
LIN {X 0,Y 560.714,Z 1101.762,A -85,B 0,C 180,E1 26707.013,E2 26707.013} C_VEL
LIN {X 0,Y 561.305,Z 1093.687,A -85,B 0,C 180,E1 26704.803,E2 26704.803} C_VEL
LIN {X 0,Y 562.376,Z 1081.912,A -85,B 0,C 180,E1 26702.087,E2 26702.087} C_VEL
LIN {X 0,Y 563.525,Z 1071.216,A -85,B 0,C 180,E1 26699.977,E2 26699.977} C_VEL
LIN {X 0,Y 564.953,Z 1059.508,A -85,B 0,C 180,E1 26697.931,E2 26697.931} C_VEL
LIN {X 0,Y 567.57,Z 1040.958,A -85,B 0,C 180,E1 26695.073,E2 26695.073} C_VEL
LIN {X 0,Y 569.923,Z 1026.432,A -85,B 0,C 180,E1 26693.083,E2 26693.083} C_VEL
LIN {X 0,Y 572.991,Z 1008.301,A -85,B 0,C 180,E1 26690.916,E2 26690.916} C_VEL
LIN {X 0,Y 575.742,Z 992.276,A -85,B 0,C 180,E1 26689.233,E2 26689.233} C_VEL
LIN {X 0,Y 578.676,Z 975.197,A -85,B 0,C 180,E1 26687.635,E2 26687.635} C_VEL
LIN {X 0,Y 582.252,Z 953.672,A -85,B 0,C 180,E1 26685.875,E2 26685.875} C_VEL
LIN {X 0,Y 585.199,Z 935.195,A -85,B 0,C 180,E1 26684.563,E2 26684.563} C_VEL
LIN {X 0,Y 588.231,Z 915.311,A -85,B 0,C 180,E1 26683.323,E2 26683.323} C_VEL
LIN {X 0,Y 591.628,Z 891.042,A -85,B 0,C 180,E1 26682.033,E2 26682.033} C_VEL
LIN {X 0,Y 594.093,Z 871.16,A -85,B 0,C 180,E1 26681.137,E2 26681.137} C_VEL
LIN {X 0,Y 596.367,Z 850.675,A -85,B 0,C 180,E1 26680.351,E2 26680.351} C_VEL
LIN {X 0,Y 598.818,Z 825.09,A -85,B 0,C 180,E1 26679.552,E2 26679.552} C_VEL
LIN {X 0,Y 600.482,Z 801.904,A -85,B 0,C 180,E1 26678.999,E2 26678.999} C_VEL
LIN {X 0,Y 601.649,Z 780.191,A -85,B 0,C 180,E1 26678.608,E2 26678.608} C_VEL
LIN {X 0,Y 609.168,Z 542.747,A -85,B 0,C 180,E1 26675.259,E2 26675.259} C_VEL
LIN {X 0,Y 614.014,Z 395.552,A -85,B 0,C 180,E1 26673.145,E2 26673.145} C_VEL
LIN {X 0,Y 613.176,Z 391.869,A -85,B 0,C 180,E1 26672.973,E2 26672.973} C_VEL
LIN {X 0,Y 603.328,Z 376.739,A -85,B 0,C 180,E1 26671.414,E2 26671.414} C_VEL
LIN {X 0,Y 592.672,Z 361.769,A -85,B 0,C 180,E1 26669.625,E2 26669.625} C_VEL
LIN {X 0,Y 584.886,Z 351.524,A -85,B 0,C 180,E1 26668.209,E2 26668.209} C_VEL
LIN {X 0,Y 581.636,Z 347,A -85,B 0,C 180,E1 26667.545,E2 26667.545} C_VEL
LIN {X 0,Y 577.077,Z 338.152,A -85,B 0,C 180,E1 26665.669,E2 26665.669} C_VEL
LIN {X 0,Y 574.522,Z 333.401,A -85,B 0,C 180,E1 26664.579,E2 26664.579} C_VEL
LIN {X 0,Y 572.325,Z 329.196,A -85,B 0,C 180,E1 26663.583,E2 26663.583} C_VEL
LIN {X 0,Y 569.601,Z 324.248,A -85,B 0,C 180,E1 26662.32,E2 26662.32} C_VEL
LIN {X 0,Y 567.478,Z 320.135,A -85,B 0,C 180,E1 26661.241,E2 26661.241} C_VEL
LIN {X 0,Y 564.841,Z 315.938,A -85,B 0,C 180,E1 26659.978,E2 26659.978} C_VEL
LIN {X 0,Y 564.162,Z 314.434,A -85,B 0,C 180,E1 26659.571,E2 26659.571} C_VEL
LIN {X 0,Y 561.923,Z 311.229,A -85,B 0,C 180,E1 26658.466,E2 26658.466} C_VEL
LIN {X 0,Y 561.463,Z 309.474,A -85,B 0,C 180,E1 26657.944,E2 26657.944} C_VEL
LIN {X 0,Y 561.436,Z 309.294,A -85,B 0,C 180,E1 26654.754,E2 26654.754} C_VEL
LIN {X 0,Y 561.425,Z 309.246,A -85,B 0,C 180,E1 26651.402,E2 26651.402} C_VEL
LIN {X 0,Y 561.42,Z 309.257,A -85,B 0,C 180,E1 26648.191,E2 26648.191} C_VEL
LIN {X 0,Y 561.429,Z 309.28,A -85,B 0,C 180,E1 26644.904,E2 26644.904} C_VEL
LIN {X 0,Y 561.431,Z 309.238,A -85,B 0,C 180,E1 26641.531,E2 26641.531} C_VEL
LIN {X 0,Y 561.431,Z 309.284,A -85,B 0,C 180,E1 26638.163,E2 26638.163} C_VEL
LIN {X 0,Y 561.42,Z 309.252,A -85,B 0,C 180,E1 26634.891,E2 26634.891} C_VEL
LIN {X 0,Y 561.424,Z 309.251,A -85,B 0,C 180,E1 26631.706,E2 26631.706} C_VEL
LIN {X 0,Y 561.431,Z 309.289,A -85,B 0,C 180,E1 26628.379,E2 26628.379} C_VEL
LIN {X 0,Y 561.424,Z 309.242,A -85,B 0,C 180,E1 26624.928,E2 26624.928} C_VEL
LIN {X 0,Y 561.43,Z 309.259,A -85,B 0,C 180,E1 26621.625,E2 26621.625} C_VEL
LIN {X 0,Y 561.421,Z 309.282,A -85,B 0,C 180,E1 26618.366,E2 26618.366} C_VEL
LIN {X 0,Y 561.51,Z 309.77,A -85,B 0,C 180,E1 26617.489,E2 26617.489} C_VEL
LIN {X 0,Y 563.18,Z 313.353,A -85,B 0,C 180,E1 26616.455,E2 26616.455} C_VEL
LIN {X 0,Y 564.806,Z 315.451,A -85,B 0,C 180,E1 26615.74,E2 26615.74} C_VEL
LIN {X 0,Y 566.829,Z 319.17,A -85,B 0,C 180,E1 26614.73,E2 26614.73} C_VEL
LIN {X 0,Y 568.018,Z 320.879,A -85,B 0,C 180,E1 26614.227,E2 26614.227} C_VEL
LIN {X 0,Y 570.262,Z 324.802,A -85,B 0,C 180,E1 26613.216,E2 26613.216} C_VEL
LIN {X 0,Y 574.106,Z 331.578,A -85,B 0,C 180,E1 26611.582,E2 26611.582} C_VEL
LIN {X 0,Y 577.061,Z 336.872,A -85,B 0,C 180,E1 26610.407,E2 26610.407} C_VEL
LIN {X 0,Y 579.905,Z 342.121,A -85,B 0,C 180,E1 26609.311,E2 26609.311} C_VEL
LIN {X 0,Y 584.339,Z 349.933,A -85,B 0,C 180,E1 26607.79,E2 26607.79} C_VEL
LIN {X 0,Y 596.683,Z 366.632,A -85,B 0,C 180,E1 26605.587,E2 26605.587} C_VEL
LIN {X 0,Y 607.183,Z 382.051,A -85,B 0,C 180,E1 26603.861,E2 26603.861} C_VEL
LIN {X 0,Y 617.465,Z 398.198,A -85,B 0,C 180,E1 26602.309,E2 26602.309} C_VEL
LIN {X 0,Y 617.825,Z 401.597,A -85,B 0,C 180,E1 26602.204,E2 26602.204} C_VEL
LIN {X 0,Y 611.492,Z 609.716,A -85,B 0,C 180,E1 26599.203,E2 26599.203} C_VEL
LIN {X 0,Y 605.696,Z 824.742,A -85,B 0,C 180,E1 26596.196,E2 26596.196} C_VEL
LIN {X 0,Y 604.316,Z 849.499,A -85,B 0,C 180,E1 26595.754,E2 26595.754} C_VEL
LIN {X 0,Y 602.138,Z 877.899,A -85,B 0,C 180,E1 26595.06,E2 26595.06} C_VEL
LIN {X 0,Y 600.152,Z 899.234,A -85,B 0,C 180,E1 26594.405,E2 26594.405} C_VEL
LIN {X 0,Y 597.959,Z 920.152,A -85,B 0,C 180,E1 26593.643,E2 26593.643} C_VEL
LIN {X 0,Y 595.748,Z 939.579,A -85,B 0,C 180,E1 26592.822,E2 26592.822} C_VEL
LIN {X 0,Y 593.242,Z 959.43,A -85,B 0,C 180,E1 26591.869,E2 26591.869} C_VEL
LIN {X 0,Y 590.137,Z 982.753,A -85,B 0,C 180,E1 26590.587,E2 26590.587} C_VEL
LIN {X 0,Y 586.606,Z 1007.041,A -85,B 0,C 180,E1 26589.036,E2 26589.036} C_VEL
LIN {X 0,Y 583.612,Z 1025.278,A -85,B 0,C 180,E1 26587.67,E2 26587.67} C_VEL
LIN {X 0,Y 580.751,Z 1042.218,A -85,B 0,C 180,E1 26586.256,E2 26586.256} C_VEL
LIN {X 0,Y 577.879,Z 1059.048,A -85,B 0,C 180,E1 26584.697,E2 26584.697} C_VEL
LIN {X 0,Y 574.971,Z 1076.249,A -85,B 0,C 180,E1 26582.928,E2 26582.928} C_VEL
LIN {X 0,Y 571.472,Z 1097.138,A -85,B 0,C 180,E1 26580.49,E2 26580.49} C_VEL
LIN {X 0,Y 569.138,Z 1111.837,A -85,B 0,C 180,E1 26578.545,E2 26578.545} C_VEL
LIN {X 0,Y 567.018,Z 1125.778,A -85,B 0,C 180,E1 26576.496,E2 26576.496} C_VEL
LIN {X 0,Y 564.885,Z 1141.381,A -85,B 0,C 180,E1 26573.912,E2 26573.912} C_VEL
LIN {X 0,Y 563.287,Z 1154.234,A -85,B 0,C 180,E1 26571.448,E2 26571.448} C_VEL
LIN {X 0,Y 562.168,Z 1164.525,A -85,B 0,C 180,E1 26569.21,E2 26569.21} C_VEL
LIN {X 0,Y 561.304,Z 1173.92,A -85,B 0,C 180,E1 26566.879,E2 26566.879} C_VEL
LIN {X 0,Y 560.6,Z 1183.955,A -85,B 0,C 180,E1 26563.933,E2 26563.933} C_VEL
LIN {X 0,Y 560.221,Z 1190.831,A -85,B 0,C 180,E1 26561.426,E2 26561.426} C_VEL
LIN {X 0,Y 560.038,Z 1196.124,A -85,B 0,C 180,E1 26559.039,E2 26559.039} C_VEL
LIN {X 0,Y 559.949,Z 1200.486,A -85,B 0,C 180,E1 26556.459,E2 26556.459} C_VEL
LIN {X 0,Y 559.913,Z 1203.505,A -85,B 0,C 180,E1 26553.686,E2 26553.686} C_VEL
LIN {X 0,Y 559.916,Z 1204.736,A -85,B 0,C 180,E1 26551.228,E2 26551.228} C_VEL
LIN {X 0,Y 559.906,Z 1204.804,A -85,B 0,C 180,E1 26549.079,E2 26549.079} C_VEL
LIN {X 0,Y 559.917,Z 1203.845,A -85,B 0,C 180,E1 26546.827,E2 26546.827} C_VEL
LIN {X 0,Y 559.934,Z 1201.534,A -85,B 0,C 180,E1 26544.364,E2 26544.364} C_VEL
LIN {X 0,Y 560.018,Z 1197.151,A -85,B 0,C 180,E1 26541.478,E2 26541.478} C_VEL
LIN {X 0,Y 560.181,Z 1191.594,A -85,B 0,C 180,E1 26538.886,E2 26538.886} C_VEL
LIN {X 0,Y 560.532,Z 1185.077,A -85,B 0,C 180,E1 26536.456,E2 26536.456} C_VEL
LIN {X 0,Y 561.163,Z 1175.941,A -85,B 0,C 180,E1 26533.649,E2 26533.649} C_VEL
LIN {X 0,Y 562.082,Z 1165.446,A -85,B 0,C 180,E1 26531.002,E2 26531.002} C_VEL
LIN {X 0,Y 563.161,Z 1155.269,A -85,B 0,C 180,E1 26528.765,E2 26528.765} C_VEL
LIN {X 0,Y 564.639,Z 1143.132,A -85,B 0,C 180,E1 26526.409,E2 26526.409} C_VEL
LIN {X 0,Y 566.812,Z 1127.181,A -85,B 0,C 180,E1 26523.72,E2 26523.72} C_VEL
LIN {X 0,Y 569.021,Z 1112.608,A -85,B 0,C 180,E1 26521.563,E2 26521.563} C_VEL
LIN {X 0,Y 571.336,Z 1097.984,A -85,B 0,C 180,E1 26519.618,E2 26519.618} C_VEL
LIN {X 0,Y 574.6,Z 1078.508,A -85,B 0,C 180,E1 26517.313,E2 26517.313} C_VEL
LIN {X 0,Y 577.784,Z 1059.604,A -85,B 0,C 180,E1 26515.356,E2 26515.356} C_VEL
LIN {X 0,Y 580.645,Z 1042.823,A -85,B 0,C 180,E1 26513.798,E2 26513.798} C_VEL
LIN {X 0,Y 583.449,Z 1026.214,A -85,B 0,C 180,E1 26512.405,E2 26512.405} C_VEL
LIN {X 0,Y 586.373,Z 1008.465,A -85,B 0,C 180,E1 26511.065,E2 26511.065} C_VEL
LIN {X 0,Y 589.809,Z 985.489,A -85,B 0,C 180,E1 26509.569,E2 26509.569} C_VEL
LIN {X 0,Y 593.151,Z 960.738,A -85,B 0,C 180,E1 26508.188,E2 26508.188} C_VEL
LIN {X 0,Y 595.798,Z 939.98,A -85,B 0,C 180,E1 26507.183,E2 26507.183} C_VEL
LIN {X 0,Y 598.171,Z 919.364,A -85,B 0,C 180,E1 26506.31,E2 26506.31} C_VEL
LIN {X 0,Y 600.538,Z 896.892,A -85,B 0,C 180,E1 26505.498,E2 26505.498} C_VEL
LIN {X 0,Y 603.112,Z 868.112,A -85,B 0,C 180,E1 26504.658,E2 26504.658} C_VEL
LIN {X 0,Y 604.774,Z 844.672,A -85,B 0,C 180,E1 26504.131,E2 26504.131} C_VEL
LIN {X 0,Y 605.97,Z 822.672,A -85,B 0,C 180,E1 26503.753,E2 26503.753} C_VEL
LIN {X 0,Y 611.86,Z 604.303,A -85,B 0,C 180,E1 26500.701,E2 26500.701} C_VEL
LIN {X 0,Y 617.584,Z 400.338,A -85,B 0,C 180,E1 26497.799,E2 26497.799} C_VEL
LIN {X 0,Y 616.842,Z 397.457,A -85,B 0,C 180,E1 26497.67,E2 26497.67} C_VEL
LIN {X 0,Y 599.696,Z 372.922,A -85,B 0,C 180,E1 26495.35,E2 26495.35} C_VEL
LIN {X 0,Y 583.727,Z 350.955,A -85,B 0,C 180,E1 26493.035,E2 26493.035} C_VEL
LIN {X 0,Y 581.648,Z 347.387,A -85,B 0,C 180,E1 26492.552,E2 26492.552} C_VEL
LIN {X 0,Y 574.256,Z 333.166,A -85,B 0,C 180,E1 26490.212,E2 26490.212} C_VEL
LIN {X 0,Y 568.84,Z 323.367,A -85,B 0,C 180,E1 26488.448,E2 26488.448} C_VEL
LIN {X 0,Y 566.234,Z 318.619,A -85,B 0,C 180,E1 26487.559,E2 26487.559} C_VEL
LIN {X 0,Y 564.317,Z 314.896,A -85,B 0,C 180,E1 26486.861,E2 26486.861} C_VEL
LIN {X 0,Y 561.72,Z 310.612,A -85,B 0,C 180,E1 26485.97,E2 26485.97} C_VEL
LIN {X 0,Y 561.445,Z 309.426,A -85,B 0,C 180,E1 26485.695,E2 26485.695} C_VEL
LIN {X 0,Y 561.431,Z 309.237,A -85,B 0,C 180,E1 26482.293,E2 26482.293} C_VEL
LIN {X 0,Y 561.437,Z 309.298,A -85,B 0,C 180,E1 26478.913,E2 26478.913} C_VEL
LIN {X 0,Y 561.422,Z 309.229,A -85,B 0,C 180,E1 26475.531,E2 26475.531} C_VEL
LIN {X 0,Y 561.425,Z 309.292,A -85,B 0,C 180,E1 26472.236,E2 26472.236} C_VEL
LIN {X 0,Y 561.431,Z 309.229,A -85,B 0,C 180,E1 26468.81,E2 26468.81} C_VEL
LIN {X 0,Y 561.435,Z 309.288,A -85,B 0,C 180,E1 26465.416,E2 26465.416} C_VEL
LIN {X 0,Y 561.42,Z 309.291,A -85,B 0,C 180,E1 26462.143,E2 26462.143} C_VEL
LIN {X 0,Y 561.437,Z 309.295,A -85,B 0,C 180,E1 26458.877,E2 26458.877} C_VEL
LIN {X 0,Y 561.432,Z 309.295,A -85,B 0,C 180,E1 26455.506,E2 26455.506} C_VEL
LIN {X 0,Y 561.418,Z 309.299,A -85,B 0,C 180,E1 26452.118,E2 26452.118} C_VEL
LIN {X 0,Y 561.438,Z 309.293,A -85,B 0,C 180,E1 26448.806,E2 26448.806} C_VEL
LIN {X 0,Y 561.413,Z 309.296,A -85,B 0,C 180,E1 26445.561,E2 26445.561} C_VEL
LIN {X 0,Y 561.43,Z 309.289,A -85,B 0,C 180,E1 26442.162,E2 26442.162} C_VEL
LIN {X 0,Y 561.445,Z 309.287,A -85,B 0,C 180,E1 26438.806,E2 26438.806} C_VEL
LIN {X 0,Y 561.397,Z 309.236,A -85,B 0,C 180,E1 26435.519,E2 26435.519} C_VEL
LIN {X 0,Y 561.445,Z 309.287,A -85,B 0,C 180,E1 26432.186,E2 26432.186} C_VEL
LIN {X 0,Y 561.41,Z 309.234,A -85,B 0,C 180,E1 26428.902,E2 26428.902} C_VEL
LIN {X 0,Y 561.405,Z 309.3,A -85,B 0,C 180,E1 26425.502,E2 26425.502} C_VEL
LIN {X 0,Y 561.439,Z 309.238,A -85,B 0,C 180,E1 26422.219,E2 26422.219} C_VEL
LIN {X 0,Y 561.489,Z 309.582,A -85,B 0,C 180,E1 26420.086,E2 26420.086} C_VEL
LIN {X 0,Y 562.795,Z 312.874,A -85,B 0,C 180,E1 26419.439,E2 26419.439} C_VEL
LIN {X 0,Y 564.059,Z 314.743,A -85,B 0,C 180,E1 26419.013,E2 26419.013} C_VEL
LIN {X 0,Y 566.09,Z 318.536,A -85,B 0,C 180,E1 26418.248,E2 26418.248} C_VEL
LIN {X 0,Y 571.656,Z 329.622,A -85,B 0,C 180,E1 26416.16,E2 26416.16} C_VEL
LIN {X 0,Y 577.632,Z 341.391,A -85,B 0,C 180,E1 26414.079,E2 26414.079} C_VEL
LIN {X 0,Y 580.694,Z 347.691,A -85,B 0,C 180,E1 26413.07,E2 26413.07} C_VEL
LIN {X 0,Y 594.228,Z 366.677,A -85,B 0,C 180,E1 26411.057,E2 26411.057} C_VEL
LIN {X 0,Y 609.772,Z 389.243,A -85,B 0,C 180,E1 26408.934,E2 26408.934} C_VEL
LIN {X 0,Y 611.271,Z 392.046,A -85,B 0,C 180,E1 26408.725,E2 26408.725} C_VEL
LIN {X 0,Y 611.994,Z 396.729,A -85,B 0,C 180,E1 26408.568,E2 26408.568} C_VEL
LIN {X 0,Y 607.703,Z 544.765,A -85,B 0,C 180,E1 26406.503,E2 26406.503} C_VEL
LIN {X 0,Y 606.8,Z 552.468,A -85,B 0,C 180,E1 26406.464,E2 26406.464} C_VEL
LIN {X 0,Y 601.866,Z 573.085,A -85,B 0,C 180,E1 26406.61,E2 26406.61} C_VEL
LIN {X 0,Y 601.158,Z 579.693,A -85,B 0,C 180,E1 26406.57,E2 26406.57} C_VEL
LIN {X 0,Y 595.09,Z 783.55,A -85,B 0,C 180,E1 26403.723,E2 26403.723} C_VEL
LIN {X 0,Y 593.589,Z 809.724,A -85,B 0,C 180,E1 26403.224,E2 26403.224} C_VEL
LIN {X 0,Y 591.574,Z 834.148,A -85,B 0,C 180,E1 26402.576,E2 26402.576} C_VEL
LIN {X 0,Y 589.452,Z 855.643,A -85,B 0,C 180,E1 26401.867,E2 26401.867} C_VEL
LIN {X 0,Y 586.615,Z 880.454,A -85,B 0,C 180,E1 26400.866,E2 26400.866} C_VEL
LIN {X 0,Y 583.759,Z 901.554,A -85,B 0,C 180,E1 26399.839,E2 26399.839} C_VEL
LIN {X 0,Y 581.05,Z 919.982,A -85,B 0,C 180,E1 26398.804,E2 26398.804} C_VEL
LIN {X 0,Y 577.907,Z 940.067,A -85,B 0,C 180,E1 26397.513,E2 26397.513} C_VEL
LIN {X 0,Y 574.194,Z 962.133,A -85,B 0,C 180,E1 26395.862,E2 26395.862} C_VEL
LIN {X 0,Y 571.195,Z 979.211,A -85,B 0,C 180,E1 26394.4,E2 26394.4} C_VEL
LIN {X 0,Y 568.191,Z 996.109,A -85,B 0,C 180,E1 26392.776,E2 26392.776} C_VEL
LIN {X 0,Y 564.703,Z 1015.626,A -85,B 0,C 180,E1 26390.631,E2 26390.631} C_VEL
LIN {X 0,Y 562.135,Z 1030.348,A -85,B 0,C 180,E1 26388.78,E2 26388.78} C_VEL
LIN {X 0,Y 559.687,Z 1044.988,A -85,B 0,C 180,E1 26386.715,E2 26386.715} C_VEL
LIN {X 0,Y 557.362,Z 1059.678,A -85,B 0,C 180,E1 26384.333,E2 26384.333} C_VEL
LIN {X 0,Y 555.174,Z 1076.559,A -85,B 0,C 180,E1 26381.216,E2 26381.216} C_VEL
LIN {X 0,Y 553.972,Z 1087.594,A -85,B 0,C 180,E1 26378.825,E2 26378.825} C_VEL
LIN {X 0,Y 553.178,Z 1096.351,A -85,B 0,C 180,E1 26376.643,E2 26376.643} C_VEL
LIN {X 0,Y 552.555,Z 1105.202,A -85,B 0,C 180,E1 26374.047,E2 26374.047} C_VEL
LIN {X 0,Y 552.205,Z 1111.987,A -85,B 0,C 180,E1 26371.556,E2 26371.556} C_VEL
LIN {X 0,Y 552.019,Z 1116.77,A -85,B 0,C 180,E1 26369.377,E2 26369.377} C_VEL
LIN {X 0,Y 551.937,Z 1120.784,A -85,B 0,C 180,E1 26366.989,E2 26366.989} C_VEL
LIN {X 0,Y 551.898,Z 1123.661,A -85,B 0,C 180,E1 26364.281,E2 26364.281} C_VEL
LIN {X 0,Y 551.917,Z 1124.783,A -85,B 0,C 180,E1 26361.981,E2 26361.981} C_VEL
LIN {X 0,Y 551.9,Z 1124.772,A -85,B 0,C 180,E1 26359.879,E2 26359.879} C_VEL
LIN {X 0,Y 551.916,Z 1123.612,A -85,B 0,C 180,E1 26357.55,E2 26357.55} C_VEL
LIN {X 0,Y 551.935,Z 1120.551,A -85,B 0,C 180,E1 26354.771,E2 26354.771} C_VEL
LIN {X 0,Y 552.015,Z 1116.922,A -85,B 0,C 180,E1 26352.611,E2 26352.611} C_VEL
LIN {X 0,Y 552.196,Z 1112.167,A -85,B 0,C 180,E1 26350.429,E2 26350.429} C_VEL
LIN {X 0,Y 552.503,Z 1105.912,A -85,B 0,C 180,E1 26348.112,E2 26348.112} C_VEL
LIN {X 0,Y 553.177,Z 1096.557,A -85,B 0,C 180,E1 26345.321,E2 26345.321} C_VEL
LIN {X 0,Y 553.982,Z 1087.567,A -85,B 0,C 180,E1 26343.079,E2 26343.079} C_VEL
LIN {X 0,Y 555.204,Z 1076.353,A -85,B 0,C 180,E1 26340.652,E2 26340.652} C_VEL
LIN {X 0,Y 557.585,Z 1058.347,A -85,B 0,C 180,E1 26337.333,E2 26337.333} C_VEL
LIN {X 0,Y 560.026,Z 1043.145,A -85,B 0,C 180,E1 26334.908,E2 26334.908} C_VEL
LIN {X 0,Y 562.413,Z 1029.105,A -85,B 0,C 180,E1 26332.938,E2 26332.938} C_VEL
LIN {X 0,Y 565.623,Z 1011.308,A -85,B 0,C 180,E1 26330.74,E2 26330.74} C_VEL
LIN {X 0,Y 568.728,Z 994.037,A -85,B 0,C 180,E1 26328.889,E2 26328.889} C_VEL
LIN {X 0,Y 571.561,Z 978.363,A -85,B 0,C 180,E1 26327.391,E2 26327.391} C_VEL
LIN {X 0,Y 575.071,Z 958.788,A -85,B 0,C 180,E1 26325.727,E2 26325.727} C_VEL
LIN {X 0,Y 578.602,Z 937.603,A -85,B 0,C 180,E1 26324.181,E2 26324.181} C_VEL
LIN {X 0,Y 581.599,Z 918.925,A -85,B 0,C 180,E1 26322.988,E2 26322.988} C_VEL
LIN {X 0,Y 584.979,Z 896.624,A -85,B 0,C 180,E1 26321.748,E2 26321.748} C_VEL
LIN {X 0,Y 588.105,Z 872.815,A -85,B 0,C 180,E1 26320.648,E2 26320.648} C_VEL
LIN {X 0,Y 590.44,Z 852.785,A -85,B 0,C 180,E1 26319.867,E2 26319.867} C_VEL
LIN {X 0,Y 592.91,Z 828.552,A -85,B 0,C 180,E1 26319.086,E2 26319.086} C_VEL
LIN {X 0,Y 594.857,Z 803.329,A -85,B 0,C 180,E1 26318.467,E2 26318.467} C_VEL
LIN {X 0,Y 596.108,Z 781.344,A -85,B 0,C 180,E1 26318.065,E2 26318.065} C_VEL
LIN {X 0,Y 604.01,Z 544.328,A -85,B 0,C 180,E1 26314.696,E2 26314.696} C_VEL
LIN {X 0,Y 609.097,Z 397.562,A -85,B 0,C 180,E1 26312.571,E2 26312.571} C_VEL
LIN {X 0,Y 604.187,Z 389.525,A -85,B 0,C 180,E1 26311.782,E2 26311.782} C_VEL
LIN {X 0,Y 593.001,Z 373.106,A -85,B 0,C 180,E1 26309.913,E2 26309.913} C_VEL
LIN {X 0,Y 582.28,Z 358.65,A -85,B 0,C 180,E1 26307.956,E2 26307.956} C_VEL
LIN {X 0,Y 574.435,Z 348.514,A -85,B 0,C 180,E1 26306.407,E2 26306.407} C_VEL
LIN {X 0,Y 573.036,Z 346.139,A -85,B 0,C 180,E1 26305.975,E2 26305.975} C_VEL
LIN {X 0,Y 569.566,Z 339.595,A -85,B 0,C 180,E1 26304.476,E2 26304.476} C_VEL
LIN {X 0,Y 567.151,Z 335.069,A -85,B 0,C 180,E1 26303.371,E2 26303.371} C_VEL
LIN {X 0,Y 564.623,Z 330.356,A -85,B 0,C 180,E1 26302.158,E2 26302.158} C_VEL
LIN {X 0,Y 562.015,Z 325.56,A -85,B 0,C 180,E1 26300.844,E2 26300.844} C_VEL
LIN {X 0,Y 559.866,Z 321.741,A -85,B 0,C 180,E1 26299.727,E2 26299.727} C_VEL
LIN {X 0,Y 557.008,Z 317.068,A -85,B 0,C 180,E1 26298.201,E2 26298.201} C_VEL
LIN {X 0,Y 556.216,Z 315.389,A -85,B 0,C 180,E1 26297.686,E2 26297.686} C_VEL
LIN {X 0,Y 553.86,Z 311.871,A -85,B 0,C 180,E1 26296.358,E2 26296.358} C_VEL
LIN {X 0,Y 553.521,Z 310.433,A -85,B 0,C 180,E1 26295.829,E2 26295.829} C_VEL
LIN {X 0,Y 553.48,Z 310.229,A -85,B 0,C 180,E1 26292.414,E2 26292.414} C_VEL
LIN {X 0,Y 553.492,Z 310.274,A -85,B 0,C 180,E1 26289.043,E2 26289.043} C_VEL
LIN {X 0,Y 553.494,Z 310.242,A -85,B 0,C 180,E1 26285.598,E2 26285.598} C_VEL
LIN {X 0,Y 553.485,Z 310.232,A -85,B 0,C 180,E1 26282.278,E2 26282.278} C_VEL
LIN {X 0,Y 553.486,Z 310.287,A -85,B 0,C 180,E1 26278.965,E2 26278.965} C_VEL
LIN {X 0,Y 553.489,Z 310.227,A -85,B 0,C 180,E1 26275.545,E2 26275.545} C_VEL
LIN {X 0,Y 553.5,Z 310.25,A -85,B 0,C 180,E1 26272.213,E2 26272.213} C_VEL
LIN {X 0,Y 553.483,Z 310.26,A -85,B 0,C 180,E1 26268.79,E2 26268.79} C_VEL
LIN {X 0,Y 553.487,Z 310.227,A -85,B 0,C 180,E1 26265.457,E2 26265.457} C_VEL
LIN {X 0,Y 553.494,Z 310.262,A -85,B 0,C 180,E1 26262.115,E2 26262.115} C_VEL
LIN {X 0,Y 553.532,Z 310.524,A -85,B 0,C 180,E1 26259.651,E2 26259.651} C_VEL
LIN {X 0,Y 555.116,Z 314.204,A -85,B 0,C 180,E1 26258.441,E2 26258.441} C_VEL
LIN {X 0,Y 556.86,Z 316.203,A -85,B 0,C 180,E1 26257.623,E2 26257.623} C_VEL
LIN {X 0,Y 558.838,Z 320.083,A -85,B 0,C 180,E1 26256.484,E2 26256.484} C_VEL
LIN {X 0,Y 560.188,Z 321.893,A -85,B 0,C 180,E1 26255.874,E2 26255.874} C_VEL
LIN {X 0,Y 562.487,Z 325.92,A -85,B 0,C 180,E1 26254.746,E2 26254.746} C_VEL
LIN {X 0,Y 563.559,Z 327.853,A -85,B 0,C 180,E1 26254.234,E2 26254.234} C_VEL
LIN {X 0,Y 566.309,Z 332.495,A -85,B 0,C 180,E1 26253.014,E2 26253.014} C_VEL
LIN {X 0,Y 569.366,Z 337.986,A -85,B 0,C 180,E1 26251.695,E2 26251.695} C_VEL
LIN {X 0,Y 572.359,Z 343.412,A -85,B 0,C 180,E1 26250.485,E2 26250.485} C_VEL
LIN {X 0,Y 575.791,Z 349.57,A -85,B 0,C 180,E1 26249.213,E2 26249.213} C_VEL
LIN {X 0,Y 582.57,Z 358.501,A -85,B 0,C 180,E1 26247.855,E2 26247.855} C_VEL
LIN {X 0,Y 592.371,Z 371.628,A -85,B 0,C 180,E1 26246.091,E2 26246.091} C_VEL
LIN {X 0,Y 603.226,Z 387.634,A -85,B 0,C 180,E1 26244.261,E2 26244.261} C_VEL
LIN {X 0,Y 612.789,Z 402.816,A -85,B 0,C 180,E1 26242.773,E2 26242.773} C_VEL
LIN {X 0,Y 605.995,Z 611.934,A -85,B 0,C 180,E1 26239.728,E2 26239.728} C_VEL
LIN {X 0,Y 599.81,Z 825.224,A -85,B 0,C 180,E1 26236.71,E2 26236.71} C_VEL
LIN {X 0,Y 598.196,Z 852.559,A -85,B 0,C 180,E1 26236.208,E2 26236.208} C_VEL
LIN {X 0,Y 596.001,Z 878.833,A -85,B 0,C 180,E1 26235.543,E2 26235.543} C_VEL
LIN {X 0,Y 593.957,Z 899.773,A -85,B 0,C 180,E1 26234.891,E2 26234.891} C_VEL
LIN {X 0,Y 591.674,Z 920.562,A -85,B 0,C 180,E1 26234.125,E2 26234.125} C_VEL
LIN {X 0,Y 589.147,Z 941.639,A -85,B 0,C 180,E1 26233.219,E2 26233.219} C_VEL
LIN {X 0,Y 585.892,Z 966.438,A -85,B 0,C 180,E1 26231.988,E2 26231.988} C_VEL
LIN {X 0,Y 582.385,Z 990.238,A -85,B 0,C 180,E1 26230.593,E2 26230.593} C_VEL
LIN {X 0,Y 579.388,Z 1009.755,A -85,B 0,C 180,E1 26229.297,E2 26229.297} C_VEL
LIN {X 0,Y 576.444,Z 1028.328,A -85,B 0,C 180,E1 26227.918,E2 26227.918} C_VEL
LIN {X 0,Y 574.032,Z 1042.221,A -85,B 0,C 180,E1 26226.749,E2 26226.749} C_VEL
LIN {X 0,Y 571.109,Z 1058.493,A -85,B 0,C 180,E1 26225.23,E2 26225.23} C_VEL
LIN {X 0,Y 568.192,Z 1074.817,A -85,B 0,C 180,E1 26223.542,E2 26223.542} C_VEL
LIN {X 0,Y 564.879,Z 1093.743,A -85,B 0,C 180,E1 26221.359,E2 26221.359} C_VEL
LIN {X 0,Y 561.878,Z 1111.064,A -85,B 0,C 180,E1 26219.065,E2 26219.065} C_VEL
LIN {X 0,Y 559.757,Z 1124.375,A -85,B 0,C 180,E1 26217.097,E2 26217.097} C_VEL
LIN {X 0,Y 557.749,Z 1137.63,A -85,B 0,C 180,E1 26214.915,E2 26214.915} C_VEL
LIN {X 0,Y 555.8,Z 1152.162,A -85,B 0,C 180,E1 26212.196,E2 26212.196} C_VEL
LIN {X 0,Y 554.441,Z 1163.605,A -85,B 0,C 180,E1 26209.708,E2 26209.708} C_VEL
LIN {X 0,Y 553.52,Z 1172.703,A -85,B 0,C 180,E1 26207.449,E2 26207.449} C_VEL
LIN {X 0,Y 552.862,Z 1180.921,A -85,B 0,C 180,E1 26205.095,E2 26205.095} C_VEL
LIN {X 0,Y 552.339,Z 1189.025,A -85,B 0,C 180,E1 26202.334,E2 26202.334} C_VEL
LIN {X 0,Y 552.079,Z 1195.294,A -85,B 0,C 180,E1 26199.591,E2 26199.591} C_VEL
LIN {X 0,Y 551.97,Z 1199.532,A -85,B 0,C 180,E1 26197.18,E2 26197.18} C_VEL
LIN {X 0,Y 551.918,Z 1202.669,A -85,B 0,C 180,E1 26194.676,E2 26194.676} C_VEL
LIN {X 0,Y 551.91,Z 1204.6,A -85,B 0,C 180,E1 26191.869,E2 26191.869} C_VEL
LIN {X 0,Y 551.895,Z 1204.872,A -85,B 0,C 180,E1 26189.377,E2 26189.377} C_VEL
LIN {X 0,Y 551.916,Z 1203.978,A -85,B 0,C 180,E1 26186.989,E2 26186.989} C_VEL
LIN {X 0,Y 551.93,Z 1201.872,A -85,B 0,C 180,E1 26184.595,E2 26184.595} C_VEL
LIN {X 0,Y 552,Z 1198.251,A -85,B 0,C 180,E1 26181.983,E2 26181.983} C_VEL
LIN {X 0,Y 552.17,Z 1192.609,A -85,B 0,C 180,E1 26179.145,E2 26179.145} C_VEL
LIN {X 0,Y 552.519,Z 1186.072,A -85,B 0,C 180,E1 26176.607,E2 26176.607} C_VEL
LIN {X 0,Y 552.999,Z 1178.801,A -85,B 0,C 180,E1 26174.264,E2 26174.264} C_VEL
LIN {X 0,Y 553.836,Z 1169.63,A -85,B 0,C 180,E1 26171.739,E2 26171.739} C_VEL
LIN {X 0,Y 555.152,Z 1157.326,A -85,B 0,C 180,E1 26168.887,E2 26168.887} C_VEL
LIN {X 0,Y 556.58,Z 1145.997,A -85,B 0,C 180,E1 26166.609,E2 26166.609} C_VEL
LIN {X 0,Y 558.322,Z 1133.823,A -85,B 0,C 180,E1 26164.432,E2 26164.432} C_VEL
LIN {X 0,Y 560.9,Z 1117.228,A -85,B 0,C 180,E1 26161.811,E2 26161.811} C_VEL
LIN {X 0,Y 563.604,Z 1100.917,A -85,B 0,C 180,E1 26159.567,E2 26159.567} C_VEL
LIN {X 0,Y 566.273,Z 1085.443,A -85,B 0,C 180,E1 26157.656,E2 26157.656} C_VEL
LIN {X 0,Y 569.654,Z 1066.711,A -85,B 0,C 180,E1 26155.586,E2 26155.586} C_VEL
LIN {X 0,Y 573.385,Z 1045.863,A -85,B 0,C 180,E1 26153.576,E2 26153.576} C_VEL
LIN {X 0,Y 576.152,Z 1030.131,A -85,B 0,C 180,E1 26152.223,E2 26152.223} C_VEL
LIN {X 0,Y 579.153,Z 1011.376,A -85,B 0,C 180,E1 26150.812,E2 26150.812} C_VEL
LIN {X 0,Y 582.144,Z 992.13,A -85,B 0,C 180,E1 26149.516,E2 26149.516} C_VEL
LIN {X 0,Y 585.231,Z 971.383,A -85,B 0,C 180,E1 26148.276,E2 26148.276} C_VEL
LIN {X 0,Y 588.936,Z 944.477,A -85,B 0,C 180,E1 26146.891,E2 26146.891} C_VEL
LIN {X 0,Y 591.684,Z 921.92,A -85,B 0,C 180,E1 26145.907,E2 26145.907} C_VEL
LIN {X 0,Y 594.036,Z 900.887,A -85,B 0,C 180,E1 26145.124,E2 26145.124} C_VEL
LIN {X 0,Y 596.142,Z 879.574,A -85,B 0,C 180,E1 26144.454,E2 26144.454} C_VEL
LIN {X 0,Y 598.24,Z 854.743,A -85,B 0,C 180,E1 26143.818,E2 26143.818} C_VEL
LIN {X 0,Y 599.986,Z 826.538,A -85,B 0,C 180,E1 26143.287,E2 26143.287} C_VEL
LIN {X 0,Y 602.333,Z 747.587,A -85,B 0,C 180,E1 26142.168,E2 26142.168} C_VEL
LIN {X 0,Y 608.581,Z 526.316,A -85,B 0,C 180,E1 26139.046,E2 26139.046} C_VEL
LIN {X 0,Y 612.131,Z 402.488,A -85,B 0,C 180,E1 26137.258,E2 26137.258} C_VEL
LIN {X 0,Y 595.584,Z 378.669,A -85,B 0,C 180,E1 26134.983,E2 26134.983} C_VEL
LIN {X 0,Y 579.599,Z 356.575,A -85,B 0,C 180,E1 26132.623,E2 26132.623} C_VEL
LIN {X 0,Y 574.229,Z 349.041,A -85,B 0,C 180,E1 26131.727,E2 26131.727} C_VEL
LIN {X 0,Y 566.638,Z 334.544,A -85,B 0,C 180,E1 26129.262,E2 26129.262} C_VEL
LIN {X 0,Y 561.047,Z 324.492,A -85,B 0,C 180,E1 26127.375,E2 26127.375} C_VEL
LIN {X 0,Y 558.545,Z 319.866,A -85,B 0,C 180,E1 26126.472,E2 26126.472} C_VEL
LIN {X 0,Y 556.599,Z 316.454,A -85,B 0,C 180,E1 26125.769,E2 26125.769} C_VEL
LIN {X 0,Y 555.439,Z 314.564,A -85,B 0,C 180,E1 26125.357,E2 26125.357} C_VEL
LIN {X 0,Y 553.681,Z 311.276,A -85,B 0,C 180,E1 26124.656,E2 26124.656} C_VEL
LIN {X 0,Y 553.519,Z 310.455,A -85,B 0,C 180,E1 26124.436,E2 26124.436} C_VEL
LIN {X 0,Y 553.495,Z 310.222,A -85,B 0,C 180,E1 26121.069,E2 26121.069} C_VEL
LIN {X 0,Y 553.491,Z 310.251,A -85,B 0,C 180,E1 26117.776,E2 26117.776} C_VEL
LIN {X 0,Y 553.481,Z 310.236,A -85,B 0,C 180,E1 26114.436,E2 26114.436} C_VEL
LIN {X 0,Y 553.488,Z 310.235,A -85,B 0,C 180,E1 26111.145,E2 26111.145} C_VEL
LIN {X 0,Y 553.501,Z 310.246,A -85,B 0,C 180,E1 26107.682,E2 26107.682} C_VEL
LIN {X 0,Y 553.482,Z 310.27,A -85,B 0,C 180,E1 26104.305,E2 26104.305} C_VEL
LIN {X 0,Y 553.498,Z 310.268,A -85,B 0,C 180,E1 26100.932,E2 26100.932} C_VEL
LIN {X 0,Y 553.488,Z 310.266,A -85,B 0,C 180,E1 26097.619,E2 26097.619} C_VEL
LIN {X 0,Y 553.48,Z 310.269,A -85,B 0,C 180,E1 26094.194,E2 26094.194} C_VEL
LIN {X 0,Y 553.5,Z 310.272,A -85,B 0,C 180,E1 26090.958,E2 26090.958} C_VEL
LIN {X 0,Y 553.476,Z 310.278,A -85,B 0,C 180,E1 26087.586,E2 26087.586} C_VEL
LIN {X 0,Y 553.489,Z 310.276,A -85,B 0,C 180,E1 26084.17,E2 26084.17} C_VEL
LIN {X 0,Y 553.502,Z 310.279,A -85,B 0,C 180,E1 26080.805,E2 26080.805} C_VEL
LIN {X 0,Y 553.468,Z 310.284,A -85,B 0,C 180,E1 26077.48,E2 26077.48} C_VEL
LIN {X 0,Y 553.488,Z 310.217,A -85,B 0,C 180,E1 26074.076,E2 26074.076} C_VEL
LIN {X 0,Y 553.497,Z 310.265,A -85,B 0,C 180,E1 26070.751,E2 26070.751} C_VEL
LIN {X 0,Y 553.457,Z 310.234,A -85,B 0,C 180,E1 26067.427,E2 26067.427} C_VEL
LIN {X 0,Y 553.499,Z 310.235,A -85,B 0,C 180,E1 26064.175,E2 26064.175} C_VEL
LIN {X 0,Y 553.49,Z 310.482,A -85,B 0,C 180,E1 26061.369,E2 26061.369} C_VEL
LIN {X 0,Y 554.903,Z 313.935,A -85,B 0,C 180,E1 26060.624,E2 26060.624} C_VEL
LIN {X 0,Y 556.294,Z 316.015,A -85,B 0,C 180,E1 26060.127,E2 26060.127} C_VEL
LIN {X 0,Y 558.351,Z 319.835,A -85,B 0,C 180,E1 26059.319,E2 26059.319} C_VEL
LIN {X 0,Y 561.459,Z 325.934,A -85,B 0,C 180,E1 26058.1,E2 26058.1} C_VEL
LIN {X 0,Y 566.443,Z 335.844,A -85,B 0,C 180,E1 26056.214,E2 26056.214} C_VEL
LIN {X 0,Y 572.248,Z 347.339,A -85,B 0,C 180,E1 26054.177,E2 26054.177} C_VEL
LIN {X 0,Y 588.488,Z 370.02,A -85,B 0,C 180,E1 26051.672,E2 26051.672} C_VEL
LIN {X 0,Y 605.278,Z 394.435,A -85,B 0,C 180,E1 26049.328,E2 26049.328} C_VEL
LIN {X 0,Y 606.482,Z 396.873,A -85,B 0,C 180,E1 26049.155,E2 26049.155} C_VEL
LIN {X 0,Y 606.512,Z 402.36,A -85,B 0,C 180,E1 26049.056,E2 26049.056} C_VEL
LIN {X 0,Y 601.158,Z 579.693,A -85,B 0,C 180,E1 26046.57,E2 26046.57} C_VEL
LIN {X 0,Y 600.249,Z 587.393,A -85,B 0,C 180,E1 26046.53,E2 26046.53} C_VEL
LIN {X 0,Y 595.3,Z 608.002,A -85,B 0,C 180,E1 26046.68,E2 26046.68} C_VEL
LIN {X 0,Y 594.576,Z 614.61,A -85,B 0,C 180,E1 26046.64,E2 26046.64} C_VEL
LIN {X 0,Y 589.332,Z 784.184,A -85,B 0,C 180,E1 26044.256,E2 26044.256} C_VEL
LIN {X 0,Y 587.762,Z 810.489,A -85,B 0,C 180,E1 26043.75,E2 26043.75} C_VEL
LIN {X 0,Y 585.687,Z 834.811,A -85,B 0,C 180,E1 26043.102,E2 26043.102} C_VEL
LIN {X 0,Y 583.536,Z 855.895,A -85,B 0,C 180,E1 26042.403,E2 26042.403} C_VEL
LIN {X 0,Y 580.591,Z 880.818,A -85,B 0,C 180,E1 26041.396,E2 26041.396} C_VEL
LIN {X 0,Y 577.626,Z 901.999,A -85,B 0,C 180,E1 26040.361,E2 26040.361} C_VEL
LIN {X 0,Y 574.683,Z 921.325,A -85,B 0,C 180,E1 26039.268,E2 26039.268} C_VEL
LIN {X 0,Y 571.081,Z 943.598,A -85,B 0,C 180,E1 26037.813,E2 26037.813} C_VEL
LIN {X 0,Y 567.403,Z 964.116,A -85,B 0,C 180,E1 26036.237,E2 26036.237} C_VEL
LIN {X 0,Y 564.309,Z 980.931,A -85,B 0,C 180,E1 26034.774,E2 26034.774} C_VEL
LIN {X 0,Y 560.812,Z 999.764,A -85,B 0,C 180,E1 26032.927,E2 26032.927} C_VEL
LIN {X 0,Y 557.43,Z 1017.493,A -85,B 0,C 180,E1 26030.913,E2 26030.913} C_VEL
LIN {X 0,Y 554.883,Z 1031.333,A -85,B 0,C 180,E1 26029.144,E2 26029.144} C_VEL
LIN {X 0,Y 552.193,Z 1046.645,A -85,B 0,C 180,E1 26026.949,E2 26026.949} C_VEL
LIN {X 0,Y 549.738,Z 1061.154,A -85,B 0,C 180,E1 26024.536,E2 26024.536} C_VEL
LIN {X 0,Y 548.05,Z 1072.272,A -85,B 0,C 180,E1 26022.432,E2 26022.432} C_VEL
LIN {X 0,Y 546.306,Z 1085.946,A -85,B 0,C 180,E1 26019.481,E2 26019.481} C_VEL
LIN {X 0,Y 545.414,Z 1094.888,A -85,B 0,C 180,E1 26017.267,E2 26017.267} C_VEL
LIN {X 0,Y 544.792,Z 1102.604,A -85,B 0,C 180,E1 26015.054,E2 26015.054} C_VEL
LIN {X 0,Y 544.299,Z 1110.553,A -85,B 0,C 180,E1 26012.316,E2 26012.316} C_VEL
LIN {X 0,Y 544.052,Z 1116.006,A -85,B 0,C 180,E1 26009.895,E2 26009.895} C_VEL
LIN {X 0,Y 543.962,Z 1119.87,A -85,B 0,C 180,E1 26007.682,E2 26007.682} C_VEL
LIN {X 0,Y 543.905,Z 1122.654,A -85,B 0,C 180,E1 26005.466,E2 26005.466} C_VEL
LIN {X 0,Y 543.913,Z 1124.605,A -85,B 0,C 180,E1 26002.819,E2 26002.819} C_VEL
LIN {X 0,Y 543.894,Z 1124.858,A -85,B 0,C 180,E1 26000.263,E2 26000.263} C_VEL
LIN {X 0,Y 543.91,Z 1124.01,A -85,B 0,C 180,E1 25998.119,E2 25998.119} C_VEL
LIN {X 0,Y 543.915,Z 1122.131,A -85,B 0,C 180,E1 25995.957,E2 25995.957} C_VEL
LIN {X 0,Y 543.989,Z 1118.696,A -85,B 0,C 180,E1 25993.448,E2 25993.448} C_VEL
LIN {X 0,Y 544.159,Z 1113.417,A -85,B 0,C 180,E1 25990.798,E2 25990.798} C_VEL
LIN {X 0,Y 544.443,Z 1107.727,A -85,B 0,C 180,E1 25988.564,E2 25988.564} C_VEL
LIN {X 0,Y 544.93,Z 1100.804,A -85,B 0,C 180,E1 25986.307,E2 25986.307} C_VEL
LIN {X 0,Y 545.811,Z 1090.952,A -85,B 0,C 180,E1 25983.614,E2 25983.614} C_VEL
LIN {X 0,Y 547.189,Z 1078.603,A -85,B 0,C 180,E1 25980.799,E2 25980.799} C_VEL
LIN {X 0,Y 549.123,Z 1065.408,A -85,B 0,C 180,E1 25978.127,E2 25978.127} C_VEL
LIN {X 0,Y 551.195,Z 1052.676,A -85,B 0,C 180,E1 25975.908,E2 25975.908} C_VEL
LIN {X 0,Y 553.596,Z 1039.02,A -85,B 0,C 180,E1 25973.8,E2 25973.8} C_VEL
LIN {X 0,Y 556.821,Z 1021.557,A -85,B 0,C 180,E1 25971.458,E2 25971.458} C_VEL
LIN {X 0,Y 559.742,Z 1006.17,A -85,B 0,C 180,E1 25969.644,E2 25969.644} C_VEL
LIN {X 0,Y 563.295,Z 987.785,A -85,B 0,C 180,E1 25967.722,E2 25967.722} C_VEL
LIN {X 0,Y 567.031,Z 967.791,A -85,B 0,C 180,E1 25965.923,E2 25965.923} C_VEL
LIN {X 0,Y 570.217,Z 950.407,A -85,B 0,C 180,E1 25964.541,E2 25964.541} C_VEL
LIN {X 0,Y 574,Z 929.121,A -85,B 0,C 180,E1 25963.052,E2 25963.052} C_VEL
LIN {X 0,Y 577.525,Z 907.006,A -85,B 0,C 180,E1 25961.739,E2 25961.739} C_VEL
LIN {X 0,Y 580.326,Z 888.115,A -85,B 0,C 180,E1 25960.769,E2 25960.769} C_VEL
LIN {X 0,Y 582.859,Z 869.317,A -85,B 0,C 180,E1 25959.933,E2 25959.933} C_VEL
LIN {X 0,Y 585.722,Z 845.563,A -85,B 0,C 180,E1 25959.04,E2 25959.04} C_VEL
LIN {X 0,Y 588.033,Z 821.053,A -85,B 0,C 180,E1 25958.316,E2 25958.316} C_VEL
LIN {X 0,Y 589.549,Z 801.285,A -85,B 0,C 180,E1 25957.854,E2 25957.854} C_VEL
